	pt^ := (pData^ / 16#10) + 48 + (((pData^ / 16#10)/10)*7);
	pt:=pt+1;
	pt^ := (pData^ AND 16#0F)  + 48 + (((pData^ AND 16#0F)/10)*7);
	pt:=pt+1;

	xl:=xl+2;

	DataLen:=DataLen-1;
	pData:=pData+1;

END_WHILE

pt^:=0;
END_FUNCTION

(* POU Plant_Objects/obj_CIR, ST *)
FUNCTION_BLOCK obj_CIR

(* === CIRCOLATORE STANDARD ===
   v1.0[16/04/15] - Versioning
   v1.1[11/08/15] - Added status reconstruction
*)
VAR CONSTANT
	SampleNr		: BYTE := 120;	(* 1 minute of observation *)
END_VAR
VAR_INPUT
	(* Settings *)
	ID				: BYTE;
	ExtStatus		: BOOL;	(* TRUE: external status signal input available, FALSE: no external status input *)

	(* Physical inputs (Force) *)
	CIR_RUN_REQ		: BOOL; (* External run request (no heat or cold requested) *)
	CIR_STOP_REQ	: BOOL; (* External stop request (has priority over RUN signals!) *)

	(* Physical inputs (Feedback) *)
	Pump_AL			: BOOL; (* Pump Alarm *)
	Pump_ST			: BOOL; (* Pump Status *)
	Pump_AUTO		: BOOL; (* Pump Auto/Manual *)

	(* Controls *)
	OnOff			: BOOL;	(* On/Off from chrono *)
	InitOK			: BOOL;

	(* Timings *)
	OnDelay		:	TIME;	(* Switch on delay *)
	OffDelay	:	TIME;	(* Switch off delay *)

	(* Input temperature needed if no real feedback about status is available *)
	Tprobe		:	INT;
END_VAR
VAR_OUTPUT
	CIR_EN			: BOOL;

	Ctrl_Run		: BOOL;		(* Logical status of the device: 0: Not running (switched off), 1: running *)
	Run				: BOOL;		(* Real status *)

	Status_Log		: WORD;
	Status_Vis		: DWORD;
END_VAR
VAR
	CIR_AUTO	: 	BOOL; (* Auto/Manual input signal *)
	Pump_En		:	BOOL;

	(* Filters *)
	fPump_ST	: 	FLT_TAP := (INITEV:=FALSE);
	fPump_En	:	FLT_EVENT;
	fCIR_AUTO	:	FLT_TAP;
	fStatus		:	FLT_EVENT;
	fStatusFault:	BOOL;

	(* Timer manage switch on/off delay *)
	Delay		: 	TONOF;

	(* Alarm and Warning counters *)
	AlarmCtr	:	BYTE;
	WarningCtr	:	BYTE;

	(* Filers on alarms and faults *)
	AlarmHw		:	FLT_TAP := (INITEV:=FALSE);

	(* Variables for status reconstruction *)
	aTprobe		:	ARRAY [1..SampleNr] OF INT;
	sample		:	BYTE;
	Tmean		:	INT;
	sum			:	INT;
	i			:	BYTE;
END_VAR
Init();

StatusRebuild();
(* Check alarms and warnings *)
CheckFault();

PumpManager();

IF AlarmCtr>0 THEN
	Status_Log := 2;
	Status_Vis := COLOR_RED;
ELSIF WarningCtr>0 OR fPump_ST.OUT THEN
	Status_Log := 1;
	Status_Vis := COLOR_YELLOW;
ELSE
	Status_Log := 0;
	Status_Vis := COLOR_GREEN;
END_IF

Lamp.UpdateStatus(obj_Status := Status_Log);
END_FUNCTION_BLOCK
ACTION AddLogData:
Logger.s1:=INSERT('&CIR=',BYTE_TO_STRING(ID),4);
IF ID<10 THEN Logger.s1:=INSERT(Logger.s1,'0',4); END_IF

Logger.s1:=CONCAT(Logger.s1,SEL(Pump_En,'0','100'));
Logger.s1:=CONCAT(Logger.s1,';');
Logger.s1:=CONCAT(Logger.s1,WORD_TO_STRING(Status_Log));
Logger.s1:=CONCAT(Logger.s1,';');
Logger.s1:=CONCAT(Logger.s1,SEL(CIR_RUN_REQ,'0','100'));
Logger.s1:=CONCAT(Logger.s1,';');
Logger.s1:=CONCAT(Logger.s1,SEL(CIR_STOP_REQ,'0','100'));


ADDSTRING(ADR(Logger.TData), ADR(Logger.s1), Logger.TLen);
END_ACTION
ACTION CheckFault:
(*** ALARMS ***)

(* Hardware alarm (physical input *)
AlarmHw(IN:=Pump_AL);

IF AlarmHw.EVH THEN
	LogEv(EL_Alarm,EO_CIR,ID,3,'');
	AlarmCtr := AlarmCtr + 1;
END_IF

IF AlarmHw.EVL THEN
	LogEv(EL_Log,EO_CIR,ID,4,'');
	AlarmCtr := SEL(AlarmCtr=0, AlarmCtr-1, 0);
END_IF

IF ExtStatus THEN
	fPump_ST(IN:=(Pump_ST<>CIR_EN));

	IF fPump_ST.EVH THEN
		IF Pump_AUTO THEN
			LogEv(SEL(Pump_ST,EL_Alarm,EL_Wrn),EO_CIR,ID,SEL(Pump_ST,5,6),'');
		ELSE
			LogEv(EL_Wrn,EO_CIR,ID,SEL(Pump_ST,1,2),'');
		END_IF
	END_IF

ELSE
	fPump_ST(IN:=fStatusFault);

	IF fPump_ST.EVH THEN
		IF Pump_AUTO THEN
			LogEv(SEL(OnOff,EL_Alarm,EL_Wrn),EO_CIR,ID,SEL(OnOff,5,6),'');
		ELSE
			LogEv(EL_Wrn,EO_CIR,ID,SEL(OnOff,1,2),'');
		END_IF
	END_IF
END_IF
END_ACTION
ACTION Init:
IF NOT InitOK THEN

	Delay.PT_OF := SEL(OffDelay=T#0ms, OffDelay, Plant_CirOffDelay);
	Delay.PT_ON := SEL(OnDelay=T#0ms, OnDelay, Plant_CirOnDelay) + WORD_TO_TIME(1000*ID);

	Pump_En := FALSE;

	InitOK := TRUE;

END_IF
END_ACTION
ACTION PumpManager:
(* Verify if in Auto or Manual mode *)
fCIR_AUTO(IN:=Pump_AUTO);

IF fCIR_AUTO.EVH THEN
	LogEv(EL_Log,EO_CIR,ID,8,'CIR_Auto');
	WarningCtr := SEL(WarningCtr=0, WarningCtr-1,0);
END_IF

(* Manual -> Keep switched on *)
IF fCIR_AUTO.EVL THEN
	LogEv(EL_Wrn,EO_CIR,ID,7,'CIR_Manual');
	WarningCtr := WarningCtr + 1;

	(* Switch on pump *)
	Pump_En := TRUE;
END_IF

(* Verify if OnOff is changed *)
Ctrl_Run := OnOff;

(* Check switch on or switch off delay *)
Delay(IN:=Ctrl_Run);

(* Do these instructions only if in AUTO mode *)
IF Pump_AUTO THEN
	(* If priority request *)
	IF CIR_STOP_REQ THEN Pump_En := FALSE;
	ELSIF CIR_RUN_REQ THEN Pump_En := TRUE;
	ELSE Pump_En := Delay.OUT;
	END_IF

	(* Set RUN signal (for external objects) *)
	IF AlarmHw.OUT THEN
		Run:=FALSE;
	ELSE
		Run:=Pump_En;
	END_IF
END_IF

(* Set value on physical outuput! *)
CIR_EN := Pump_En;
END_ACTION
ACTION StatusRebuild:
IF NOT ExtStatus THEN
	(* Check every 20 seconds *)
	IF  sample<sampleNr THEN
	
		aTprobe[sample] := Tprobe;
		sample := sample + 1;
	
	ELSE
	
		SHIFT_ARRAY(ADR(aTprobe),SampleNr);
	
		FOR i:=1 TO SampleNr BY 1 DO
			sum := sum + aTprobe[i];
		END_FOR
	
		Tmean := sum/SampleNr;
	
		(* CIR should be on but revealed temperature is decreasing *)
		IF OnOff AND (Tprobe<aTprobe[1]) THEN
			fStatusFault := TRUE;
		ELSE
			fStatusFault := FALSE;
		END_IF
	
		(* CIR should be off but revealed temperature is increasing *)
		IF NOT OnOff AND (Tprobe>aTprobe[1]) THEN
			fStatusFault := TRUE;
		ELSE
			fStatusFault := FALSE;
		END_IF
	END_IF
END_IF
END_ACTION

(* POU Utils Functions/TONOF, ST *)
FUNCTION_BLOCK TONOF
VAR_INPUT
	IN		: BOOL;
	PT_ON	: TIME; (* time to pass, before OUT is set *)
	PT_OF	: TIME; (* time to pass, before OUT is reset *)
END_VAR
VAR_OUTPUT
	OUT		: BOOL;
END_VAR
VAR
	timer	: TON;
END_VAR
IF IN<>OUT THEN
	timer(IN:=TRUE,PT:=SEL(IN,PT_OF,PT_ON));
	IF timer.Q THEN OUT:=IN; END_IF
ELSE
	timer(IN:=FALSE);
END_IF
END_FUNCTION_BLOCK

(* POU Plant_Objects/obj_CRON_EDITOR, ST *)
FUNCTION_BLOCK obj_CRON_EDITOR
(* === EDITOR CRONOGRAFO ===
   v1.0[16/04/15] - Versioning
   v1.1[19/05/15] - Create empty profile when not found
*)
VAR_INPUT

	(* Common selections *)
	CN_Sel:			BYTE:=1;
	CN_Act:			BYTE;
	CN_YSel:		WORD:=2015;
	CN_YAct:		WORD;

	(* Profile editor *)
	PR_Sel: 		BYTE:=1;
	PR_Act:			BYTE;
	PR_TT:			REAL;
	PR:				typ_Cron_Profile;
	(* Profile signals *)
	PR_Load:		BOOL;
	PR_Save:		BOOL;

	(* Calendar editor *)
	CA_Sel:			BYTE:=1; (* Calendar month selected *)
	CA_Act:			BYTE;    (* Calendar month active *)
	CA_DayF:		BYTE:=0;
	CA_DayL:		BYTE:=31;
	CA_TPR:			BYTE;
	CA:				typ_Cron_Calendar; (* Only used for first 32 entries *)
	(* Calendar signals *)
	CA_Load:		BOOL;
	CA_Save:		BOOL;

	(* Jolly editor *)
	JL:				ARRAY[0..9] OF typ_Cron_Jolly;
	(* Jolly signals *)
	JL_Load:		BOOL;
	JL_Save:		BOOL;

END_VAR
VAR_OUTPUT
	Message		: STRING;
END_VAR
VAR
	sFileName	: STRING;
	sFileMode	: STRING;
	hFile		: DWORD;
	Buf			: ARRAY[0..512] OF BYTE; (* AVOID THIS!! *)

	i			: WORD;
	ver			: BYTE;
	r1			: BOOL;
	r2			: DWORD;

END_VAR
IF PR_Load THEN PR_Load_Exe(); PR_Load:=FALSE; END_IF
IF PR_Save THEN PR_Save_Exe(); PR_Save:=FALSE; END_IF
IF CA_Load THEN CA_Load_Exe(); CA_Load:=FALSE; END_IF
IF CA_Save THEN CA_Save_Exe(); CA_Save:=FALSE; END_IF
IF JL_Load THEN JL_Load_Exe(); JL_Load:=FALSE; END_IF
IF JL_Save THEN JL_Save_Exe(); JL_Save:=FALSE; END_IF
END_FUNCTION_BLOCK
ACTION CA_Load_Exe:
sFileMode:='r';
FileOpen();

IF hFile<>0 THEN

	(* Read calendar month *)
	FOR i := 0 TO 31 DO
		r1:=SysFileSetPos(File:=hFile, Pos:=(1024 + ((CA_Sel-1)*32 + i)*4));
		r2:=SysFileRead(File:=hFile, Buffer:=ADR(CA.Profile[i]), Size:=1);
	END_FOR

	(* Close file *)
	SysFileClose(File:=hFile);

	(* Validate data *)
	CA_Act :=CA_Sel;
	CN_Act :=CN_Sel;
	CN_YAct:=CN_YSel;

	Message:='Calendar load OK';

END_IF
END_ACTION
ACTION CA_Save_Exe:
sFileMode:='a';
FileOpen();

IF hFile<>0 THEN

	(* Write calendar month *)
	FOR i := 0 TO 31 DO
		r1:=SysFileSetPos(File:=hFile, Pos:=(1024 + ((CA_Sel-1)*32 + i)*4));
		r2:=SysFileGetPos(hFile);
		r2:=SysFileWrite(File:=hFile, Buffer:=ADR(CA.Profile[i]), Size:=1);
	END_FOR

	(* Close file *)
	SysFileClose(File:=hFile);

	Message:='Calendar save OK';

END_IF
END_ACTION
ACTION FileOpen:
(* Create current filename 'yyyyCRnn.DAT' *)
sFileName:=CONCAT(FilesPath,WORD_TO_STRING(CN_YSel));
sFileName:=CONCAT(STR1:=sFileName, STR2:='CR');
IF CN_Sel<10 THEN
sFileName:=CONCAT(STR1:=sFileName, STR2:='0');
END_IF
sFileName:=CONCAT(STR1:=sFileName, STR2:=BYTE_TO_STRING(CN_Sel));
sFileName:=CONCAT(STR1:=sFileName, STR2:='.DAT');

(* Check file version and size! *)
(* ... *)

(* Open data file *)
hFile:=SysFileOpen(FileName:=sFileName, Mode:='r');

(* File not found *)
IF hFile=0 THEN
	Message:='File not found - created empty file';
	(* Create empty file *)
	hFile:=SysFileOpen(FileName:=sFileName, Mode:='w');
	MEMCLR(pDestinationAddress:=ADR(Buf), BytesToClear:=SIZEOF(Buf));
	FOR i := 0 TO 10239 BY 512 DO
		SysFileWrite(File:=hFile, Buffer:=ADR(Buf), Size:=512);
	END_FOR
	Buf[0]:=1;
	SysFileSetPos(File:=hFile, Pos:=0);
	SysFileWrite(File:=hFile, Buffer:=ADR(Buf), Size:=1);
END_IF

(* Close file *)
SysFileClose(File:=hFile);

(* Open data file *)
hFile:=SysFileOpen(FileName:=sFileName, Mode:=sFileMode);
END_ACTION
ACTION JL_Load_Exe:
sFileMode:='r';
FileOpen();

IF hFile<>0 THEN

	(* Read jolly *)
	r1:=SysFileSetPos(File:=hFile, Pos:=512);
	r2:=SysFileRead(File:=hFile, Buffer:=ADR(JL), Size:=SIZEOF(JL));

	(* Close file *)
	SysFileClose(File:=hFile);

	(* Validate data *)
	CN_Act:=CN_Sel;
	CN_YAct:=CN_YSel;

	Message:='Jolly load OK';

END_IF
END_ACTION
ACTION JL_Save_Exe:
sFileMode:='a';
FileOpen();

IF hFile<>0 THEN

	(* Write selected profile *)
	r1:=SysFileSetPos(File:=hFile, Pos:=512);
	r2:=SysFileWrite(File:=hFile, Buffer:=ADR(JL), Size:=SIZEOF(JL));

	(* Close file *)
	SysFileClose(File:=hFile);

	Message:='Jolly save OK';

END_IF
END_ACTION
ACTION PR_Load_Exe:
sFileMode:='r';
FileOpen();

IF hFile<>0 THEN

	(* Read selected profile *)
	r1:=SysFileSetPos(File:=hFile, Pos:=(3072 + 512*PR_Sel));
	r2:=SysFileRead(File:=hFile, Buffer:=ADR(PR), Size:=SIZEOF(PR));

	(* Close file *)
	SysFileClose(File:=hFile);

	(* Validate data *)
	PR_Act:=PR_Sel;
	CN_Act:=CN_Sel;
	CN_YAct:=CN_YSel;

	Message:='Profile load OK';

END_IF
END_ACTION
ACTION PR_Save_Exe:
sFileMode:='a';
FileOpen();

IF hFile<>0 THEN

	(* Write selected profile *)
	r1:=SysFileSetPos(File:=hFile, Pos:=(3072 + 512*PR_Sel));
	r2:=SysFileWrite(File:=hFile, Buffer:=ADR(PR), Size:=SIZEOF(PR));

	(* Close file *)
	SysFileClose(File:=hFile);

	Message:='Profile save OK';

END_IF
END_ACTION

(* POU Plant_Objects/obj_CRONTER, ST *)
FUNCTION_BLOCK obj_CRONTER
(* === THERMOSTAT ===
   v1.0[30/07/15] - Versioning
*)
VAR_INPUT
	(* Settings *)
	ID			: BYTE;		(* Index of instanced object *)

	InitOK		: BOOL;
	Alarm		: BOOL;
	Warning		: BOOL;

	Profile		: typ_Cron_Profile; 				(* Profilo attivo *)
	ProfileNr	: BYTE;								(* Indice profilo attivo *)
	CalendarIdx : WORD;								(* Indice calendario attivo *)
	Jolly		: ARRAY[0..9] OF typ_Cron_Jolly;	(* Jolly attivi *)

	Temperature	: INT;
	Local_MaxRunTAmb	:	INT;					(* Local maximum environment temperature, NOT "TAMB" *)


	Histeresys:INT; (* isteresi per la ripartenza del Comando ON*)


END_VAR
VAR_IN_OUT
END_VAR
VAR_OUTPUT
	SetPoint		: INT;
	Run				: BOOL;
	AntifreezeForce	: BOOL;

	(* Status *)
	Status_Log		: BYTE;
	Status_Vis 		: DWORD;
END_VAR
VAR
	Buf: 	ARRAY[0..512] OF BYTE; (* AVOID THIS!! *)
	hFile: 	DWORD;
	sFile: 	STRING;
	sFile2: STRING;

	i:		WORD;
	t1:		DWORD;
	t2:		BOOL;

END_VAR
(* Check initialization *)
IF NOT InitOK THEN Init(); END_IF

(* Check Temperature *)
IF Temperature < 400(*Local_MaxRunTAmb*) THEN

	(* LOCAL environment temperature lower than maximum allowed -> Proceed with SetPoint adjustment *)
	(* Chrono *)
	IF CalendarIdx<>Sys.Time_CT_Day THEN DB_Load(); END_IF
	SetPoint:=Profile.Setpoint[Sys.Time_CT_Quarter];

	(* Check jolly *)
	FOR i := 0 TO 9 DO
		IF ( DT_TO_DWORD(Jolly[i].Start)>0  AND Jolly[i].End>Jolly[i].Start AND
		     Jolly[i].Start<=Sys.Time_CT_DT AND Jolly[i].End>Sys.Time_CT_DT ) THEN
				SetPoint:=Jolly[i].Temp;
		END_IF
	END_FOR

(*
	IF SetPoint < 180 THEN
		(* Switch off the device *)
		Run := FALSE;
	ELSE
		(* Set according to feedback T - Histeresys of 1°C *)
		IF Temperature >= (SetPoint + 5) THEN
			Run := FALSE;
		ELSIF Temperature <= (SetPoint - 5) THEN
			Run := TRUE;
		END_IF

		(* Between "SetPoint-5" and "SetPoint+5" last state (ON or OFF) of "Run" is kept	*)
	END_IF
*)
(*	IF SetPoint>0 THEN Run := TRUE;
	ELSIF SetPoint=0 THEN Run := FALSE;
	END_IF *)

		IF Temperature >= (SetPoint) THEN
			Run := FALSE;
		ELSIF Temperature <= (SetPoint - Histeresys) THEN
			Run := TRUE;
		END_IF




ELSE
	(* Environment overtemperature: stop heating -> Stop device *)
	Run := FALSE;
END_IF

(* Freeze warning: Switch on and heat! *)
(*IF Temperature < Plant_AntiFreezeTAmb THEN AntifreezeForce := TRUE;
ELSE AntifreezeForce := FALSE;
END_IF*)



(* Status color *)
   IF Alarm   THEN Status_Log:=2; Status_Vis:=COLOR_RED;
ELSIF Warning THEN Status_Log:=1; Status_Vis:=COLOR_YELLOW;
              ELSE Status_Log:=0; Status_Vis:=COLOR_GREEN;
			  END_IF
END_FUNCTION_BLOCK
ACTION AddLogData:
Logger.s1:=INSERT('&THER=',BYTE_TO_STRING(ID),5);
IF ID<10 THEN Logger.s1:=INSERT(Logger.s1,'0',5); END_IF

Logger.s1:=CONCAT(Logger.s1,INT_TO_STRING(SetPoint));			Logger.s1:=CONCAT(Logger.s1,';');

Logger.s1:=CONCAT(Logger.s1,WORD_TO_STRING(Status_Log));
ADDSTRING(ADR(Logger.TData), ADR(Logger.s1), Logger.TLen);
END_ACTION
ACTION DB_Create:
(* Create empty file *)
hFile:=SysFileOpen(FileName:=sFile, Mode:='w');

MEMCLR(pDestinationAddress:=ADR(Buf), BytesToClear:=SIZEOF(Buf));
FOR i := 0 TO 10239 BY 512 DO
	t1:=SysFileWrite(File:=hFile, Buffer:=ADR(Buf), Size:=512);		(* Clear created file (all bytes 0) *)
END_FOR
Buf[0]:=1;
t2:=SysFileSetPos(File:=hFile, Pos:=0);
t1:=SysFileWrite(File:=hFile, Buffer:=ADR(Buf), Size:=1);
SysFileClose(File:=hFile);
END_ACTION
ACTION DB_Load:
DB_SetName();

(* Open data file *)
hFile:=SysFileOpen(FileName:=sFile, Mode:='r');

(* File not found *)
IF hFile=0 THEN
	Warning:=TRUE;
	LogEv(EL_Wrn,EO_CRON,ID,1,'No_data_file');
	DB_Create();
	(* Reopen file *)
	hFile:=SysFileOpen(FileName:=sFile, Mode:='r');
	IF hfile=0 THEN
		Alarm:=TRUE;
		LogEv(EL_Alarm,EO_CRON,ID,3,'Filesystem_error');
		RETURN;
	END_IF
END_IF

(* Check version *)
SysFileRead(File:=hFile, Buffer:=ADR(Buf), Size:=1);
IF Buf[0]<>1 THEN
	IF NOT Alarm THEN
		Alarm:=TRUE;
		LogEv(EL_Alarm,EO_CRON,ID,2,'Bad_data_version');
	END_IF
	SysFileClose(File:=hFile);
	RETURN;
END_IF

(* Read Jolly data *)
t2:=SysFileSetPos(File:=hFile, Pos:=512);
t1:=SysFileRead(File:=hFile, Buffer:=ADR(Jolly), Size:=SIZEOF(Jolly));
(* Read active profile index *)
CalendarIdx:=Sys.Time_CT_Day;
t2:=SysFileSetPos(File:=hFile, Pos:=(1024+4*CalendarIdx));
t1:=SysFileRead(File:=hFile, Buffer:=ADR(ProfileNr), Size:=SIZEOF(ProfileNr));
(* Read active profile *)
t2:=SysFileSetPos(File:=hFile, Pos:=(3072+512*ProfileNr));
t1:=SysFileRead(File:=hFile, Buffer:=ADR(Profile), Size:=SIZEOF(Profile));

(* Close file and validate data *)
SysFileClose(File:=hFile);
END_ACTION
ACTION DB_SetName:
(* Create current filename 'yyyyCRnn.DAT' *)
sFile:=CONCAT(FilesPath,WORD_TO_STRING(Sys.Time_Year));
sFile:=CONCAT(STR1:=sFile, STR2:='CR');
IF ID<10 THEN
sFile:=CONCAT(STR1:=sFile, STR2:='0');
END_IF
sFile:=CONCAT(STR1:=sFile, STR2:=BYTE_TO_STRING(ID));
sFile:=CONCAT(STR1:=sFile, STR2:='.DAT');
END_ACTION
ACTION Init:
DB_Load();
InitOK:=TRUE;
END_ACTION

(* POU Plant_Objects/obj_CTL, ST *)
FUNCTION_BLOCK obj_CTL
(* === PULSE VOLUME COUNTER ===
   v1.0[16/04/15] - Versioning
*)
VAR_INPUT
	(* Settings *)
	ID				: BYTE;	(* Index of instanced object *)
	Peso			: DWORD;
	(* Physical inputs *)
	CTL_ST			: BOOL;
END_VAR
VAR_IN_OUT
	COUNT			: DWORD;
END_VAR
VAR_OUTPUT
	(* Status *)
	Status_Log		: BYTE;
END_VAR
VAR
	Filter			: FLT_TAP := ( INITEV:=FALSE );
	Filter01			: FLT_TAP := ( INITEV:=FALSE );
	Timer			: TON;
	TCount			: DWORD;
	TCount01		: DWORD;
	i				: DWORD;

	TempoSicurezzaPerdita: DINT;
	TimerConataLitriPerdita:TOF;


	MorenoTest: BOOL;
	erroreTest: BOOL;
END_VAR

VAR_INPUT RETAIN
	LimiteMaxPerdita: INT;
END_VAR
(* Execute timer *)
Timer(IN:=NOT Timer.Q, PT:=T#60m);

(* Execute filter on counter status *)
Filter(IN:=CTL_ST);
Filter01(IN:=CTL_ST);


(*

(* Count event *)
IF Filter.EVH THEN
	COUNT:=COUNT+Peso;

	TCount:=TCount+1;
	(* Check flow rate *)
	IF TCount>=Plant_MaxWaterLoss THEN


		i:=(TCount*TIME_TO_DWORD(Timer.PT))/TIME_TO_DWORD(Timer.ET);	(* Estimated mc per hour *)
		i:= i * Peso;

		(* NB The weight is multiplied by 10 -> Need to divide it by 10 server side *)
		LogEv(EL_AlarmStop,EO_CTL,ID,1,DWORD_TO_STRING(i));
		Status_Log:=2;

		TCount:=0;
		Timer(IN:=FALSE);
	END_IF
END_IF
(* Check timer *)
IF Timer.Q THEN
	TCount:=0;							(* One hour is elapsed *)
	IF TCount<Plant_MaxWaterLoss THEN
		Status_Log:=0;
	END_IF
END_IF

*)


(*** calcolo del tempo del contalitri minimo per la segnalazione dell'allarme perdita *****)

(* il limiteMAXPerdita è espresso in l/h con n.1 decimale, Quindi dividendolo per il peso dell'impulso e per 60minuti, otteniamo
quanto tempo deve passare minimo fra un impulsao e l'altro *)

LimiteMaxPerdita:=LIMIT(LimiteMaxPerdita,10,LimiteMaxPerdita+1);
TempoSicurezzaPerdita:=3600000/((LimiteMaxPerdita/peso)); (* espresso in ms *)

IF Filter01.EVH THEN
(*	COUNT:=COUNT+Peso; *)

	TCount01:=TCount01+1;
	IF TimerConataLitriPerdita.Q AND NOT erroreTest THEN

		(* NB The weight is multiplied by 10 -> Need to divide it by 10 server side *)

		LogEv(EL_AlarmStop,EO_CTL,ID,1,CONCAT('LimiteMAXPerdita_l/h>',DWORD_TO_STRING(LimiteMaxPerdita/10)));
		Status_Log:=2;

		erroreTest:=TRUE;
		TimerConataLitriPerdita(IN:=FALSE, PT:= t#1s, Q=> , ET=> );
	END_IF


	IF NOT TimerConataLitriPerdita.Q AND erroreTest THEN
		erroreTest:=FALSE;
		TCount01:=0;
		Status_Log:=0;
	END_IF

END_IF





TimerConataLitriPerdita(IN:=Filter01.EVH, PT:= DINT_TO_TIME(TempoSicurezzaPerdita), Q=> , ET=> );
END_FUNCTION_BLOCK
ACTION AddLogData:
Logger.s1:=INSERT('&CTL=',BYTE_TO_STRING(ID),4);
IF ID<10 THEN Logger.s1:=INSERT(Logger.s1,'0',4); END_IF

Logger.s1:=CONCAT(Logger.s1,DWORD_TO_STRING(COUNT));			Logger.s1:=CONCAT(Logger.s1,';');

Logger.s1:=CONCAT(Logger.s1,WORD_TO_STRING(Status_Log));
ADDSTRING(ADR(Logger.TData), ADR(Logger.s1), Logger.TLen);
END_ACTION

(* POU Plant_Objects/obj_MBUS, ST *)
FUNCTION_BLOCK obj_MBUS
(* === M-BUS PROTOCOL INTERFACE ===
   v1.0[16/03/15] - Added interface errors
*)
VAR_INPUT
	(* Settings *)
	ID				: BYTE;
	COM				: BYTE;
	BAUDRATE		: COM_BAUDRATE;
	(* Interface *)
	MBus 			: typMBus;
	MBus_Master 	: FbMBusMaster;
END_VAR
VAR_OUTPUT
	(* Status *)
	Status_Log		: BYTE;
	Status_Vis 		: DWORD;
END_VAR
VAR
	Alarm			: FLT_EVENT;
END_VAR
MBus_Master( bCOMPORT:=COM , enumBAUDRATE:=BAUDRATE , utMBus:=MBus );

(* Check status *)
Alarm(IN:=(MBus.bCOM_ERROR<>0));
IF Alarm.EVH THEN
	LogEv(EL_Alarm,EO_MBUS,ID,1,BYTE_TO_STRING(MBus.bCOM_ERROR));
END_IF
IF Alarm.EVL THEN
	LogEv(EL_Log,EO_MBUS,ID,2,'MBUS_OK');
END_IF

(* Log/visu status *)
   IF Alarm.IN   					THEN Status_Log:=2; Status_Vis:=COLOR_RED;
ELSIF (MBus.bL1_ERROR AND 16#1F)<>0 THEN Status_Log:=1; Status_Vis:=COLOR_YELLOW;
  				 					ELSE Status_Log:=0; Status_Vis:=COLOR_GREEN;
END_IF
END_FUNCTION_BLOCK

(* POU Plant_Objects/obj_MBUS_CTB_SHARKY775, ST *)
FUNCTION_BLOCK obj_MBUS_CTB_SHARKY775
(* === M-BUS CONTABILIZER SHARKY 775 ===
   v1.0[16/03/15] - Error management
*)
VAR_INPUT
	(* Settings *)
	ID				: BYTE;
	ADDRESS			: DWORD;
	Refresh_Period	: TIME:=t#3m;
	(* Controls *)
	Refresh_Auto	: BOOL:=TRUE; (* Enable automatic refresh *)
	Refresh_Now		: BOOL; 	  (* Force an immediate refresh *)
END_VAR
VAR_IN_OUT
	(* Interface *)
	MBUS			: obj_MBUS;
END_VAR
VAR_OUTPUT
	M1				: FbMBus_Heat;
	(* Status *)
	Status_Log		: BYTE;
	Status_Vis 	 	: DWORD;
END_VAR
VAR
	dly 	 	: TON := (PT:=t#5s);
	M1_Start	: BOOL;

	init_st		: BOOL;
	bus_st0		: BYTE;
	dev_st0		: BYTE;

(*	S1			: FbMBusSend;
	S1_Start	: BOOL;*)
(*	C1			: FbUnitConverter; *)

END_VAR
(* Auto refresh timer *)
dly(IN:=NOT (dly.Q OR Refresh_Now OR (NOT Refresh_Auto)));
(* Trigger refresh *)
IF dly.Q OR Refresh_Now THEN
	dly.PT:=Refresh_Period;
	Refresh_Now:=FALSE;
	(* Start reading *)
	M1.dwAdr:= ADDRESS;
	M1.xSND_NKE:=TRUE;
	M1_Start:=TRUE;
END_IF

(* Contabilizer module *)
M1(	utMBus:=MBUS.MBus, xStart:=M1_Start );

(* Extra actions *)
(*C1( utMBus:=MBUS.MBus, xStart:=C1_Start );*)

(* Check status *)
IF NOT init_st OR M1.bError<>bus_st0 OR M1.utMBInfo.bMStatus<>dev_st0 THEN
	init_st:=TRUE;
	bus_st0:=M1.bError; dev_st0:=M1.utMBInfo.bMStatus;
	IF bus_st0<>0 THEN
		LogEv(EL_Alarm,EO_CTB,ID,2,BYTE_TO_STRING(bus_st0));
		Status_Log:=2; Status_Vis:=COLOR_RED;
	ELSE
		IF dev_st0<>0 THEN
			Status_Log:=2; Status_Vis:=COLOR_RED;
			CASE dev_st0 OF
				16#08: LogEv(EL_Alarm,EO_CTB,ID,10,'C-1');
				16#04: LogEv(EL_Alarm,EO_CTB,ID,10,'E-8');
				16#28: LogEv(EL_Alarm,EO_CTB,ID,10,'E-4');
				16#50: LogEv(EL_Alarm,EO_CTB,ID,10,'E-1');
				16#70: LogEv(EL_Alarm,EO_CTB,ID,10,'E-7');
				16#84: LogEv(EL_Alarm,EO_CTB,ID,10,'E-9');
				16#B0: LogEv(EL_Wrn  ,EO_CTB,ID,10,'E-3');
				16#D0: LogEv(EL_Wrn  ,EO_CTB,ID,10,'E-6');
				16#F0: LogEv(EL_Alarm,EO_CTB,ID,10,'Leak');
				16#10: LogEv(EL_Wrn  ,EO_CTB,ID,10,'E-5'); Status_Log:=1; Status_Vis:=COLOR_YELLOW;
			ELSE
				LogEv(EL_Alarm,EO_CTB,ID,10,BYTE_TO_STRING(dev_st0));
			END_CASE
		ELSE
			Status_Log:=0; Status_Vis:=16#20F020;
			LogEv(EL_Log,EO_CTB,ID,1,'');
		END_IF
	END_IF
END_IF

Lamp.obj_Status := Status_Log;
Lamp.UpdateStatus();
END_FUNCTION_BLOCK
ACTION AddLogData:
Logger.s1:=INSERT('&CTB=',BYTE_TO_STRING(ID),4);
IF ID<10 THEN Logger.s1:=INSERT(Logger.s1,'0',4); END_IF

Logger.s1:=CONCAT(Logger.s1,M1.utFTemp.Value);		Logger.s1:=CONCAT(Logger.s1,';');
Logger.s1:=CONCAT(Logger.s1,M1.utRTemp.Value);		Logger.s1:=CONCAT(Logger.s1,';');
Logger.s1:=CONCAT(Logger.s1,M1.utFlow.Value);		Logger.s1:=CONCAT(Logger.s1,';');
Logger.s1:=CONCAT(Logger.s1,M1.utPower.Value);		Logger.s1:=CONCAT(Logger.s1,';');
Logger.s1:=CONCAT(Logger.s1,M1.utEnergy.Value);		Logger.s1:=CONCAT(Logger.s1,';');

Logger.s1:=CONCAT(Logger.s1,BYTE_TO_STRING(Status_Log));
ADDSTRING(ADR(Logger.TData), ADR(Logger.s1), Logger.TLen);
END_ACTION

(* POU Plant_Objects/obj_MODBUS, ST *)
FUNCTION_BLOCK obj_MODBUS
(* === MODBUS PROTOCOL INTERFACE ===
   v1.1[19/06/15] - Added new VARS allocation and searching
*)
VAR CONSTANT
	VARS_Max	: BYTE := 32;
END_VAR
VAR_INPUT
	(* Settings *)
	ID			: BYTE;
	COM			: BYTE;
	BAUDRATE	: COM_BAUDRATE;
	RS485		: BOOL := FALSE;

	(* Interface *)
	MB_MASTER	: MODBUS_EXTENDED_MASTER;
	MB_Start	: BOOL;
	MB_Query	: typModbusExtendedQuery;
	MB_Resp		: typModbusResponse;
	MB_Lock		: BOOL;

	(* Variables management *)
	VARS_En		: BOOL;
	VARS		: ARRAY [0..VARS_Max] OF typ_MODBUS_VAR;
	VARS_Check	: BOOL;
	VARS_Alarm	: BOOL;

	(* Variables allocation *)
	VAR_Pointer : POINTER TO ARRAY[0..99] OF WORD;
	VAR_Cfg		: POINTER TO typ_MODBUS_VAR;
END_VAR
VAR_OUTPUT
	(* Status *)
	Status_Log	: BYTE;
	Status_Vis	: DWORD;
END_VAR
VAR
	sta         : BYTE :=0;
	i			: BYTE;
	j			: BYTE;
	Alarm		: FLT_EVENT;
	
	VarTmr		: TON := (PT:=T#1s);
	VarSta		: BYTE; (* Status *)
	VarCnt		: BYTE; (* Scan counter *)
	VarRetry	: BYTE;
	VarAlarm	: BYTE; (* Last variable with errors *)
END_VAR
MB_MASTER(ENABLE:=TRUE,	ASCII_Mode:=FALSE, bCOM_PORT:=COM, cbCOM_BAUDRATE:=BAUDRATE, cpCOM_PARITY:=PARITY_NO,
		csCOM_STOPBITS:=STOPBITS_1,	cbsCOM_BYTESIZE:=BS_8, cfCOM_FLOW_CONTROL:=SEL(RS485,NO_FLOW_CONTROL,HALFDUPLEX),
		tTIME_OUT:=t#250ms,	StartFunction:=MB_Start, ExtQuery:=MB_Query, Response:=MB_Resp);

(* Process variable management *)
IF VARS_En THEN VARS_Process(); END_IF

(* Check status *)
Alarm(IN:=(MB_MASTER.bInterfaceError<>0));
IF Alarm.EVH THEN
	LogEv(SEL(MB_MASTER.bInterfaceError<>3,EL_Wrn,EL_Alarm),EO_MODBUS,ID,1,BYTE_TO_STRING(MB_MASTER.bInterfaceError));
END_IF
IF Alarm.EVL THEN								(* Trigger a fall edge: MODBUS back working *)
	LogEv(EL_Log,EO_MODBUS,ID,2,'MODBUS_OK');
END_IF

(* Log/visu status *)
   IF Alarm.IN   THEN Status_Log:=2; Status_Vis:=COLOR_RED;
ELSIF Vars_Alarm THEN Status_Log:=1; Status_Vis:=COLOR_YELLOW;
  				 ELSE Status_Log:=0; Status_Vis:=COLOR_GREEN;
END_IF
END_FUNCTION_BLOCK
ACTION VAR_Search:
(* Search VAR with specific pointer if not found return first free VAR
	[Last VAR is not active... used as safe area...] 
*)
j:=VARS_Max;
FOR i := 0 TO VARS_Max-1 DO
	IF VARS[i].Variable=0 AND j>i THEN j:=i; END_IF
	IF VARS[i].Variable=VAR_Pointer THEN
		VAR_Cfg:=ADR(VARS[i]);
		RETURN;
	END_IF
END_FOR
VAR_Cfg:=ADR(VARS[j]);
END_ACTION
ACTION VARS_Process:
(* Update var timers *)
VarTmr(IN:=(NOT VarTmr.Q));
IF VarTmr.Q THEN
	FOR i := 0 TO VARS_Max DO
		IF VARS[i].Refresh_Cnt>0 THEN VARS[i].Refresh_Cnt:=VARS[i].Refresh_Cnt-1; END_IF
	END_FOR
	VARS_Check:=TRUE;
END_IF


(* Process status *)
CASE VarSta OF
	0: (* === Init *)
		VarCnt:=0;
		VarSta:=1;

	1: (* === Wait check signal *)
		IF VARS_Check THEN				(* Decremented "Refresh_Cnt" *)
			VARS_Check:=FALSE;
			VarCnt:=0;
			VarSta:=2;
		END_IF

	2: (* === Check loop *)
		IF NOT (MB_Lock OR MB_Start) THEN
			WHILE VarCnt<=(VARS_Max-1) AND VarSta=2 DO
				(* Check only active vars *)
				IF VARS[VarCnt].Variable<>0 THEN			(* "Variable" is a pointer to word, so if 0 no address *)
					(* Check var auto-refresh on timer checks *)
					IF VARS[VarCnt].Refresh_Time>0 AND VARS[VarCnt].Refresh_Cnt=0 THEN
						VARS[VarCnt].Refresh_Cnt:=VARS[VarCnt].Refresh_Time;
						VarSta:=3;
					END_IF
					(* Check refresh for change or request *)
					CASE VARS[VarCnt].FunCode OF
						5,6,15,16: (* Write functions *)
							IF VARS[VarCnt].Variable_Size=1 THEN
								IF VARS[VarCnt].Variable^<>VARS[VarCnt].Variable_Mirror THEN
									VARS[VarCnt].Variable_Mirror:=VARS[VarCnt].Variable^;
									VarSta:=3;
								END_IF
							ELSE
								IF VARS[VarCnt].Variable_Mirror<>0 THEN
									VARS[VarCnt].Variable_Mirror:=0;
									VarSta:=3;
								END_IF
							END_IF
						1,2,3,4: (* Read functions *)
							IF VARS[VarCnt].Variable_Mirror<>0 THEN
								VARS[VarCnt].Variable_Mirror:=0;
								VarSta:=3;
							END_IF
					END_CASE
				END_IF
				(* Process query *)
				IF VarSta=3 THEN
					MB_Lock:=TRUE;
					MB_Query.SlaveAddress:=VARS[VarCnt].SlaveAddress;
					MB_Query.FunctionCode:=VARS[VarCnt].FunCode;
					CASE VARS[VarCnt].FunCode OF
						16#5,16#6,16#F,16#10:
							MB_Query.Read_Quantity:=0;
							MB_Query.Read_StartAddress:=0;
							MB_Query.Write_StartAddress:=VARS[VarCnt].FunAddress;
							MB_Query.Write_Quantity:=VARS[VarCnt].Variable_Size;
							IF VARS[VarCnt].Variable_Size=200 THEN
								COPY_32SWAP16(VARS[VarCnt].Variable, ADR(MB_Query.Write_Data[0]));
							ELSIF VARS[VarCnt].Variable_Size>1 THEN
								MEMCPY(VARS[VarCnt].Variable, ADR(MB_Query.Write_Data[0]), 2*VARS[VarCnt].Variable_Size);
							ELSE
								MB_Query.Write_Data[0]:=VARS[VarCnt].Variable^;
							END_IF
						16#1,16#2,16#3,16#4:
							MB_Query.Read_StartAddress:=VARS[VarCnt].FunAddress;
							IF VARS[VarCnt].Variable_Size=200 THEN MB_Query.Read_Quantity:=2; ELSE
							  MB_Query.Read_Quantity:=VARS[VarCnt].Variable_Size;
							END_IF
							MB_Query.Write_StartAddress:=0;
							MB_Query.Write_Quantity:=0;
					END_CASE
					VarRetry:=0;
					MB_Start:=TRUE;
				ELSE
					VarCnt:=VarCnt+1;
				END_IF
			END_WHILE
			(* Check loop completed -> no actions *)
			IF VarSta=2 THEN VarSta:=1; END_IF
		END_IF

	3: (* === Wait & process MB response *)
		IF NOT MB_Start THEN
			IF MB_MASTER.MB_Error=0 THEN
				CASE VARS[VarCnt].FunCode OF
					1,2,3,4:
						IF VARS[VarCnt].Variable_Size=200 THEN
							COPY_32SWAP16(ADR(MB_Resp.Data), VARS[VarCnt].Variable);
						ELSIF VARS[VarCnt].Variable_Size>1 THEN
							MEMCPY(ADR(MB_Resp.Data), VARS[VarCnt].Variable, 2*VARS[VarCnt].Variable_Size);
						ELSE
							VARS[VarCnt].Variable^:=MB_Resp.Data[0];
						END_IF
				END_CASE
				MB_Lock:=FALSE;
				(* Signal error recovery *)
				IF VARS_Alarm=TRUE AND VarCnt=VarAlarm THEN
					LogEv(EL_Wrn,EO_MODBUS,ID,5,'');
					VARS_Alarm:=FALSE;
				END_IF
				(* Next var *)
				VarCnt:=VarCnt+1;
				VarSta:=2;
			ELSE
				IF VarRetry<3 THEN
					VarRetry:=VarRetry+1;
					MB_Start:=TRUE;
				ELSE
					MB_Lock:=FALSE;
					(* Signal error *)
					IF VARS_Alarm=FALSE THEN
						LogEv(EL_Wrn,EO_MODBUS,ID,3,INT_TO_STRING(MB_MASTER.MB_Error));
						VARS_Alarm:=TRUE;
						VarAlarm:=VarCnt-1;
					END_IF
					(* Next var *)
					VarCnt:=VarCnt+1;
					VarSta:=2;
				END_IF
			END_IF
		END_IF

ELSE
	VarSta:=0;
END_CASE
END_ACTION

(* POU Plant_Objects/obj_MODBUS_CIR, ST *)
FUNCTION_BLOCK obj_MODBUS_CIR
VAR CONSTANT
	WAIT_STATE		:	BYTE := 0;
	PUMP_STATUS		:	BYTE := 1;
	PUMP_DATA		:	BYTE := 2;
	PUMP_ALARMS		:	BYTE := 3;
	PUMP_END_READ	:	BYTE := 4;
	CIR_ON_OFF		:	BYTE := 90;
	CIR_ON_OFF_CHECK:	BYTE := 91;
	CIR_END_WRITE	:	BYTE := 92;
	ERROR_STATE		:	BYTE := 100;
END_VAR
VAR_INPUT
	ID		:	BYTE;
	Address :	BYTE;		(* Pump address *)

	(* Physical inputs *)
	CIR_RUN_REQ		: BOOL; (* External run request (no heat or cold requested) *)
	CIR_STOP_REQ	: BOOL; (* External stop request (has priority over RUN signals!) *)

	Pump_AL			: BOOL; (* Alarm input signal *)
	Pump_AUTO		: BOOL;	(* Automatic/Manual input *)

	(* Controls *)
	OnOff		: 	BOOL;
	InitOK		:	BOOL;

	(* Timings *)
	OnDelay		:	TIME;
	OffDelay	:	TIME;

	(* Modbus *)
	Refresh_Now	:	BOOL;	(* Start immediately modbus state machine *)
	retryErrMax	:	BYTE := 15;
END_VAR
VAR_IN_OUT
	ModBus		:	obj_MODBUS;
END_VAR
VAR_OUTPUT
	Ctrl_Run	:	BOOL;		(* Logical status of the device: 0: Not running (switched off), 1: running *)
	Run			:	BOOL;		(* Real status *)

	Status_Log	:	WORD;
	Status_Vis	:	DWORD;
END_VAR
VAR
	Pump_En		:	WORD;

	(* Filters *)
	fPump_AL	:	FLT_TAP := (INITEV:=FALSE);
	fPump_ST	:	FLT_TAP := (INITEV:=FALSE);
	fPump_En	:	FLT_EVENT;
	fCIR_AUTO	:	FLT_TAP;
	fStatus		:	FLT_EVENT;
	fStatusFault:	BOOL;

	(* Timer manage switch on/off delay *)
	Delay		: 	TONOF;

	(* CIR data structure *)
	DataPump	:	typ_MODBUS_CIR;

	(* Modbus variables *)
	state		:	BYTE;
	retry		:	BYTE;
	retryErr	:	BYTE;
	ReadTmr		:	TON := (PT:=T#5s);
	fModbusAlr	: 	BOOL;

	(* Alarm and Warning counters *)
	AlarmCtr	:	BYTE;
	WarningCtr	:	BYTE;

	(* Filers on alarms and faults *)
	AlarmHw		:	FLT_TAP;(* := (INITEV:=FALSE);*)
	Alarm		:	FLT_EVENT := (INITEV:=FALSE);
	Inverter	:	FLT_EVENT := (INITEV:=FALSE);
	ModbusAlr	:	FLT_EVENT := (INITEV:=FALSE);

	OldAlarm	:	WORD;

	TimeOutModBus: TON;
END_VAR
Init();

(* Check alarm and warning for both pumps *)
CheckFault();

PumpManager();

(* State machine to read pump parameters *)
Stm();

IF AlarmCtr>0 THEN
	Status_Log := 2;
	Status_Vis := COLOR_RED;
ELSIF WarningCtr>0 OR fPump_ST.OUT THEN
	Status_Log := 1;
	Status_Vis := COLOR_YELLOW;
ELSE
	Status_Log := 0;
	Status_Vis := COLOR_GREEN;
END_IF

(* Update error lamp status *)
Lamp.UpdateStatus(obj_Status:=Status_Log);
END_FUNCTION_BLOCK
ACTION AddLogData:
Logger.s1:=INSERT('&CIRM=',BYTE_TO_STRING(ID),5);
IF ID<10 THEN Logger.s1:=INSERT(Logger.s1,'0',5); END_IF

(* NB If value equals 0x7FFF (32767) this means that it is not available -->> Change it to 0 *)
Logger.s1:=CONCAT(Logger.s1,WORD_TO_STRING(DataPump.PumpStatus));											Logger.s1:=CONCAT(Logger.s1,';');
Logger.s1:=CONCAT(Logger.s1,INT_TO_STRING(SEL(DataPump.PumpBoardTemp=16#7FFF,DataPump.PumpBoardTemp,0)));	Logger.s1:=CONCAT(Logger.s1,';');
Logger.s1:=CONCAT(Logger.s1,WORD_TO_STRING(SEL(DataPump.PumpVoltage=16#7FFF,DataPump.PumpVoltage,0)));		Logger.s1:=CONCAT(Logger.s1,';');
Logger.s1:=CONCAT(Logger.s1,WORD_TO_STRING(SEL(DataPump.PumpCurrent=16#7FFF,DataPump.PumpCurrent,0)));		Logger.s1:=CONCAT(Logger.s1,';');
Logger.s1:=CONCAT(Logger.s1,WORD_TO_STRING(SEL(DataPump.PumpPower=16#7FFF,DataPump.PumpPower,0)));			Logger.s1:=CONCAT(Logger.s1,';');
Logger.s1:=CONCAT(Logger.s1,WORD_TO_STRING(SEL(DataPump.PumpRPM=16#7FFF,DataPump.PumpRPM,0)));				Logger.s1:=CONCAT(Logger.s1,';');
Logger.s1:=CONCAT(Logger.s1,WORD_TO_STRING(SEL(DataPump.PumpHead=16#7FFF,DataPump.PumpHead,0)));				Logger.s1:=CONCAT(Logger.s1,';');
Logger.s1:=CONCAT(Logger.s1,WORD_TO_STRING(SEL(DataPump.PumpFlow=16#7FFF,DataPump.PumpFlow,0)));				Logger.s1:=CONCAT(Logger.s1,';');
Logger.s1:=CONCAT(Logger.s1,WORD_TO_STRING(SEL(DataPump.PumpLiqTemp=16#7FFF,DataPump.PumpLiqTemp,0)));		Logger.s1:=CONCAT(Logger.s1,';');
Logger.s1:=CONCAT(Logger.s1,DWORD_TO_STRING(SEL(DataPump.PumpOpTime=16#7FFF,DataPump.PumpOpTime,0)));		Logger.s1:=CONCAT(Logger.s1,';');


Logger.s1:=CONCAT(Logger.s1,WORD_TO_STRING(Status_Log));
Logger.s1:=CONCAT(Logger.s1,';');

Logger.s1:=CONCAT(Logger.s1,SEL(DataPump.PumpFault,'0','100'));
Logger.s1:=CONCAT(Logger.s1,';');
Logger.s1:=CONCAT(Logger.s1,SEL(CIR_RUN_REQ,'0','100'));
Logger.s1:=CONCAT(Logger.s1,';');
Logger.s1:=CONCAT(Logger.s1,SEL(CIR_STOP_REQ,'0','100'));

ADDSTRING(ADR(Logger.TData), ADR(Logger.s1), Logger.TLen);
END_ACTION
ACTION CheckFault:
(*** WARNINGS ***)

(* Verify ModBus error	*)
ModbusAlr(IN:=fModbusAlr);

IF ModbusAlr.EVH THEN
	LogEv(EL_Wrn,EO_CIRM,ID,13,SEL(ModBus.MB_MASTER.MB_Error<>0,'0','1'));
	WarningCtr := WarningCtr + 1;
END_IF

IF ModbusAlr.EVL THEN WarningCtr := SEL(WarningCtr=0, WarningCtr-1, 0); END_IF


(*** ALARMS ***)

(* Hardware alarm (physical input *)
AlarmHw(IN:=Pump_AL);

IF AlarmHw.EVH THEN
	LogEv(EL_Alarm,EO_CIRM,ID,3,'CIR_Alarm');
	AlarmCtr := AlarmCtr + 1;
END_IF

IF AlarmHw.EVL THEN
	LogEv(EL_Log,EO_CIRM,ID,4,'CIR_Alarm_Recovered');
	AlarmCtr := SEL(AlarmCtr=0, AlarmCtr-1, 0);
END_IF

(*
(* General alarm (read by Modbus) *)
Alarm(IN:=(DataPump.PumpAlarm[0] <> OldAlarm));

IF Alarm.EVH THEN
	IF DataPump.PumpAlarm[0] = 0 THEN
		LogEv(EL_Log,EO_CIRM,ID,12,'Alarm_Recovered');
		AlarmCtr := SEL(AlarmCtr=0, AlarmCtr-1, 0);
	ELSE
		LogEv(EL_Alarm,EO_CIRM,ID,11,WORD_TO_STRING(DataPump.PumpAlarm[0]));
		AlarmCtr := AlarmCtr + 1;
	END_IF

	OldAlarm := DataPump.PumpAlarm[0];
END_IF


(* Inverter pump error *)
Inverter(IN:=DataPump.PumpFault);

IF Inverter.EVH THEN
	LogEv(EL_Alarm,EO_CIRM,ID,9,'Inverter_Fault');
	AlarmCtr := AlarmCtr + 1;
END_IF

IF Inverter.EVL THEN
	LogEv(EL_Alarm,EO_CIRM,ID,10,'Inverter_Fault_Recovered');
		AlarmCtr := SEL(AlarmCtr=0, AlarmCtr-1, 0);
END_IF

*)
END_ACTION
ACTION Init:
IF NOT InitOK THEN

	Delay.PT_OF := SEL(OffDelay=T#0ms, OffDelay, Plant_CirOffDelay);
	Delay.PT_ON := SEL(OnDelay=T#0ms, OnDelay, Plant_CirOnDelay) + WORD_TO_TIME(1000*ID);

	ReadTmr.PT := WORD_TO_TIME(1000*ID);	(* 1s delay between reads of 2 different double CIRs *)

	Pump_En := 1;
	Refresh_Now := TRUE;

	InitOK := TRUE;

END_IF
END_ACTION
ACTION PumpManager:
(*** Verify Status ***)
IF Pump_AUTO THEN
	IF (Pump_En=1 AND DataPump.PumpStatus=2) OR (Pump_En=0 AND DataPump.PumpStatus=0) THEN fStatusFault := TRUE;
	ELSE fStatusFault := FALSE;
	END_IF
END_IF

fPump_ST(IN:=fStatusFault);

IF fPump_ST.EVH THEN
	LogEv(SEL(Pump_En=1,EL_Alarm,EL_Wrn),EO_CIRM,ID,SEL(Pump_En=1,5,6),'');
	WarningCtr := WarningCtr + 1;
END_IF

IF fPump_ST.EVL THEN WarningCtr := SEL(WarningCtr=0, WarningCtr-1, 0); END_IF

(* Verify if in Auto or Manual mode *)
fCIR_AUTO(IN:=Pump_AUTO);

(* Automatic *)
IF fCIR_AUTO.EVH THEN
	LogEv(EL_Log,EO_CIRM,ID,8,'CIR_Auto');
	WarningCtr := SEL(WarningCtr=0, WarningCtr-1, 0);

	Refresh_Now := TRUE;
END_IF

(* Manual -> Keep switched on *)
IF fCIR_AUTO.EVL THEN
	LogEv(EL_Wrn,EO_CIRM,ID,7,'CIR_Manual');
	WarningCtr := WarningCtr + 1;

	Pump_En := 0;
	Refresh_Now := TRUE;
END_IF

(* Verify if OnOff is changed *)
Ctrl_Run := OnOff;

(* Check switch on or switch off delay *)
Delay(IN:=Ctrl_Run);

IF Pump_AUTO THEN
	(* If priority request *)
	IF CIR_STOP_REQ THEN Pump_En := 1;
	ELSIF CIR_RUN_REQ THEN Pump_En := 0;
	ELSE Pump_En := BOOL_TO_WORD(NOT Delay.OUT);
	END_IF

	(* Set RUN signal (for external objects) *)
	IF AlarmHw.OUT THEN
		Run:=FALSE;
	ELSE
		Run:=SEL(Pump_En=1,TRUE,FALSE);
	END_IF
END_IF

(* Check if a pump enable update (modbus write) is requested *)
fPump_En(IN:=(Pump_En=1));

IF fPump_En.EVH OR fPump_En.EVL THEN
	Refresh_Now := TRUE;
END_IF
END_ACTION
ACTION Stm:
CASE state OF
	WAIT_STATE:	(* Refresh time manager *)
		ReadTmr(IN:=NOT ReadTmr.Q);
		IF ReadTmr.Q OR Refresh_Now  THEN
			state := PUMP_STATUS;
			ReadTmr.PT := T#1m;
			Refresh_Now := FALSE;
		END_IF

	(**** READ CIR PARAMETERS ****)

	PUMP_STATUS:	(* Status and Fault *)
		Modbus.MB_Lock := TRUE;
		Modbus.MB_Query.SlaveAddress := Address;
		Modbus.MB_Query.FunctionCode := 3;
		ModBus.MB_Query.Read_StartAddress := 201;
		ModBus.MB_Query.Read_Quantity := 2;
		ModBus.MB_Start := TRUE;

		state := PUMP_DATA;

	PUMP_DATA:	(* Pump data *)
		IF NOT ModBus.MB_Start AND ModBus.MB_Resp.SlaveAddress=Address  THEN
			IF ModBus.MB_MASTER.bInterfaceError<>0 THEN (*OR ModBus.MB_MASTER.MB_Error<>0 THEN*)
				state := ERROR_STATE;
			ELSE
				DataPump.PumpStatus := ModBus.MB_Resp.Data[0];
				DataPump.PumpFault	:= WORD_TO_BOOL(ModBus.MB_Resp.Data[1]);

				ModBus.MB_Query.Read_StartAddress := 210;
				ModBus.MB_Query.Read_Quantity := 12;
				ModBus.MB_Start := TRUE;

				state := PUMP_ALARMS;
			END_IF
		END_IF

	PUMP_ALARMS: (* Historical alarms *)
		IF NOT ModBus.MB_Start AND ModBus.MB_Resp.SlaveAddress=Address  THEN
			IF ModBus.MB_MASTER.bInterfaceError<>0 THEN (*OR ModBus.MB_MASTER.MB_Error<>0 THEN*)
				state := ERROR_STATE;
			ELSE
				DataPump.PumpBoardTemp 	:= WORD_TO_INT(ModBus.MB_Resp.Data[0]);
				DataPump.PumpVoltage	:= ModBus.MB_Resp.Data[2];
				DataPump.PumpCurrent	:= ModBus.MB_Resp.Data[3];
				DataPump.PumpRPM		:= ModBus.MB_Resp.Data[5];
				DataPump.PumpPower		:= ModBus.MB_Resp.Data[6];
				DataPump.PumpOpTime		:= BUILD_16TO32(ADR(ModBus.MB_Resp.Data[7]));
				DataPump.PumpHead		:= ModBus.MB_Resp.Data[9];
				DataPump.PumpFlow		:= ModBus.MB_Resp.Data[10];
				DataPump.PumpLiqTemp	:= WORD_TO_INT(ModBus.MB_Resp.Data[11]);


				ModBus.MB_Query.Read_StartAddress := 230;
				ModBus.MB_Query.Read_Quantity := 1;(*15;*)
				ModBus.MB_Start := TRUE;

				state := PUMP_END_READ;
			END_IF
		END_IF

	PUMP_END_READ:	(* Read alarms *)
		IF NOT ModBus.MB_Start AND ModBus.MB_Resp.SlaveAddress=Address  THEN
			IF ModBus.MB_MASTER.bInterfaceError<>0 THEN (*OR ModBus.MB_MASTER.MB_Error<>0 THEN*)
				state := ERROR_STATE;
			ELSE
				DataPump.PumpAlarm[0] := ModBus.MB_Resp.Data[0];	(* Read just last (most recent) alarm *)
				(*DataPump.PumpAlarm[1] := ModBus.MB_Resp.Data[1];
				DataPump.PumpAlarm[2] := ModBus.MB_Resp.Data[2];
				DataPump.PumpAlarm[3] := ModBus.MB_Resp.Data[3];
				DataPump.PumpAlarm[4] := ModBus.MB_Resp.Data[4];
				DataPump.PumpAlarm[5] := ModBus.MB_Resp.Data[5];
				DataPump.PumpAlarm[6] := ModBus.MB_Resp.Data[6];
				DataPump.PumpAlarm[7] := ModBus.MB_Resp.Data[7];
				DataPump.PumpAlarm[8] := ModBus.MB_Resp.Data[8];
				DataPump.PumpAlarm[9] := ModBus.MB_Resp.Data[9];
				DataPump.PumpAlarm[10] := ModBus.MB_Resp.Data[10];
				DataPump.PumpAlarm[11] := ModBus.MB_Resp.Data[11];
				DataPump.PumpAlarm[12] := ModBus.MB_Resp.Data[12];
				DataPump.PumpAlarm[13] := ModBus.MB_Resp.Data[13];
				DataPump.PumpAlarm[14] := ModBus.MB_Resp.Data[14];*)

				state := CIR_ON_OFF;

			END_IF
		END_IF

	(**** WRITE ON/OFF REGISTER AND VERIFY RIGHT SETTING ****)
	CIR_ON_OFF:	(* Pump On/off *)

		Modbus.MB_Query.SlaveAddress := Address;
		Modbus.MB_Query.FunctionCode := 6;
		ModBus.MB_Query.Write_StartAddress := 110;
		ModBus.MB_Query.Write_Quantity := 1;
		ModBus.MB_Query.Write_Data[0] := Pump_En;
		ModBus.MB_Start := TRUE;

		state := CIR_END_WRITE;

	CIR_END_WRITE:
		IF NOT ModBus.MB_Start THEN
			IF ModBus.MB_MASTER.bInterfaceError<>0 THEN (*OR ModBus.MB_MASTER.MB_Error<>0 THEN*)
				state := ERROR_STATE;
			ELSE
				IF fModbusAlr THEN fModbusAlr := FALSE; END_IF

				ModBus.MB_Lock := FALSE;
				retryErr := 0;
				retry := 0;
				state := WAIT_STATE;
			END_IF
		END_IF


	(**** CHECK MODBUS ERROR ****)
	ERROR_STATE: 	(* Release MODBUS *)
			MODBUS.MB_Lock:=FALSE;

			(* Retries *)
			retry:=retry+1;
			IF retry>3 THEN
				retry:=0;

				(* Verify if slave is dead *)
				IF retryErr < retryErrMaX THEN
					retryErr := retryErr + 1;
				ELSE
					fModbusAlr := TRUE;
				END_IF

				Refresh_Now := FALSE;
			END_IF

			state:=WAIT_STATE;
END_CASE

(* Controllo Time Out Ciclo ModBus *)

TimeOutModBus(In:=state<>0,PT:=t#2s);
IF TimeOutModBus.Q THEN State:=0; END_IF
END_ACTION

(* POU Plant_Objects/obj_MODBUS_CIR_DOPPIO_new, ST *)
FUNCTION_BLOCK obj_MODBUS_CIR_DOPPIO_new
VAR CONSTANT
	WAIT_STATE		:	BYTE := 0;
	PUMP1_STATUS	:	BYTE := 1;
	PUMP1_DATA		:	BYTE := 2;
	PUMP1_ALARMS	:	BYTE := 3;
	PUMP1_END_READ	:	BYTE := 4;
	PUMP2_STATUS	:	BYTE := 5;
	PUMP2_DATA		:	BYTE := 6;
	PUMP2_ALARMS	:	BYTE := 7;
	PUMP2_END_READ	:	BYTE := 8;
	CIR_ON_OFF1		:	BYTE := 90;
	CIR_ON_OFF2		:	BYTE := 91;
	CIR_ON_OFF_CHECK:	BYTE := 92;
	CIR_END_WRITE	:	BYTE := 93;
	ERROR_STATE		:	BYTE := 100;

END_VAR
VAR_INPUT
	ID		:	BYTE;
	Address1:	BYTE;		(* Pump 1 Modbus address *)
	Address2:	BYTE;		(* Pump 2 Modbus address *)

	(* Physical inputs (Force) *)
	CIR_RUN_REQ		: BOOL; (* External run request (no heat or cold requested) *)
	CIR_STOP_REQ	: BOOL; (* External stop request (has priority over RUN signals!) *)

	(* Physical inputs (Feedback) *)
	PumpA_AL		: BOOL; (* Alarm input signal *)
	PumpB_AL		: BOOL;
	PumpA_AUTO		: BOOL;	(* Automatic/Manual input *)
	PumpB_AUTO		: BOOL;

	(* Controls *)
	OnOff		: 	BOOL;	(* On/Off from chrono *)
	Mode		:	BYTE;	(* Working mode: 0-Both pumps works simultaneously, 1-Alternate every 24h, 2-Master/Backup *)
	InitOK		:	BOOL;

	(* Timings *)
	OnDelay		:	TIME;	(* Switch on delay *)
	OffDelay	:	TIME;	(* Switch off delay *)

	(* Modbus *)
	Refresh_Now	:	BOOL;	(* Start immediately modbus state machine *)
	retryErrMax	:	BYTE := 15;
END_VAR
VAR_IN_OUT
	ModBus		:	obj_MODBUS;
END_VAR
VAR_OUTPUT
	Ctrl_Run	:	BOOL;		(* Logical status of the device: 0: Not running (switched off), 1: running *)
	Run			:	BOOL;		(* Real status *)

	Status_Log	:	WORD;
	Status_Vis	:	DWORD;
END_VAR
VAR
	Status		:	BOOL;
	Pump_En		:	ARRAY [1..2] OF WORD;		(* Pumps enable *)

	ChangeTmr	: 	TON := (PT:=T#24h);			(* Timer that counts change time when in alternate mode *)
	ActivePump	: 	BYTE := 1;						(* Actual active pump *)
	NewActivePump	: BYTE := 1;

	(* Filters *)
	fPump_ST	: 	ARRAY [1..2] OF FLT_TAP := (INITEV:=FALSE);
	fPump_En	:	ARRAY [1..2] OF FLT_EVENT;
	fCIR_AUTO	:	ARRAY [1..2] OF FLT_TAP;
	fStatusFault:	ARRAY [1..2] OF BOOL;
	fBackup		:	FLT_EVENT := (INITEV:=FALSE);

	(* Timer manage switch on/off delay *)
	Delay		: 	TONOF;

	(* CIR data structure *)
	DataPump1	:	typ_MODBUS_CIR;
	DataPump2	:	typ_MODBUS_CIR;

	(* Modbus variables *)
	state		:	BYTE;
	retry		:	BYTE;
	retryErr	:	BYTE;
	ReadTmr		:	TON := (PT:=T#5s);
	fModbusAlr	: 	BOOL;

	(* Alarm and Warning counters *)
	AlarmCtr	:	BYTE;
	WarningCtr	:	BYTE;

	(* Filers on alarms and faults *)
	AlarmHw		:	ARRAY [1..2] OF FLT_TAP := (INITEV:=FALSE);
	Alarm		:	ARRAY [1..2] OF FLT_EVENT := (INITEV:=FALSE);
	Inverter	:	ARRAY [1..2] OF FLT_EVENT := (INITEV:=FALSE);
	ModbusAlr	:	FLT_EVENT := (INITEV:=FALSE);

	OldAlarmPump1	:	WORD;
	OldAlarmPump2	:	WORD;

	TimeOutModBus: TON;
END_VAR
Init();

(* Check alarm and warning for both pumps *)
CheckFault();

PumpManager();

(* State machine to read pump parameters *)
Stm();

IF AlarmCtr>0 THEN
	Status_Log := 2;
	Status_Vis := COLOR_RED;
ELSIF WarningCtr>0 THEN
	Status_Log := 1;
	Status_Vis := COLOR_YELLOW;
ELSE
	Status_Log := 0;
	Status_Vis := COLOR_GREEN;
END_IF

(* Update error lamp status *)
Lamp.UpdateStatus(obj_Status := Status_Log);
END_FUNCTION_BLOCK
ACTION AddLogData:
Logger.s1:=INSERT('&CIRDM=',BYTE_TO_STRING(ID),6);
IF ID<10 THEN Logger.s1:=INSERT(Logger.s1,'0',6); END_IF

Logger.s1:=CONCAT(Logger.s1,WORD_TO_STRING(Mode));						Logger.s1:=CONCAT(Logger.s1,';');
(* PUMP 1 *)
(* NB If value equals 0x7FFF (32767) this means that it is not available -->> Change it to 0 *)
Logger.s1:=CONCAT(Logger.s1,WORD_TO_STRING(DataPump1.PumpStatus));											Logger.s1:=CONCAT(Logger.s1,';');
Logger.s1:=CONCAT(Logger.s1,INT_TO_STRING(SEL(DataPump1.PumpBoardTemp=16#7FFF,DataPump1.PumpBoardTemp,0)));	Logger.s1:=CONCAT(Logger.s1,';');
Logger.s1:=CONCAT(Logger.s1,WORD_TO_STRING(SEL(DataPump1.PumpVoltage=16#7FFF,DataPump1.PumpVoltage,0)));		Logger.s1:=CONCAT(Logger.s1,';');
Logger.s1:=CONCAT(Logger.s1,WORD_TO_STRING(SEL(DataPump1.PumpCurrent=16#7FFF,DataPump1.PumpCurrent,0)));		Logger.s1:=CONCAT(Logger.s1,';');
Logger.s1:=CONCAT(Logger.s1,WORD_TO_STRING(SEL(DataPump1.PumpPower=16#7FFF,DataPump1.PumpPower,0)));			Logger.s1:=CONCAT(Logger.s1,';');
Logger.s1:=CONCAT(Logger.s1,WORD_TO_STRING(SEL(DataPump1.PumpRPM=16#7FFF,DataPump1.PumpRPM,0)));				Logger.s1:=CONCAT(Logger.s1,';');
Logger.s1:=CONCAT(Logger.s1,WORD_TO_STRING(SEL(DataPump1.PumpHead=16#7FFF,DataPump1.PumpHead,0)));				Logger.s1:=CONCAT(Logger.s1,';');
Logger.s1:=CONCAT(Logger.s1,WORD_TO_STRING(SEL(DataPump1.PumpFlow=16#7FFF,DataPump1.PumpFlow,0)));				Logger.s1:=CONCAT(Logger.s1,';');
Logger.s1:=CONCAT(Logger.s1,WORD_TO_STRING(SEL(DataPump1.PumpLiqTemp=16#7FFF,DataPump1.PumpLiqTemp,0)));		Logger.s1:=CONCAT(Logger.s1,';');
Logger.s1:=CONCAT(Logger.s1,DWORD_TO_STRING(SEL(DataPump1.PumpOpTime=16#7FFF,DataPump1.PumpOpTime,0)));		Logger.s1:=CONCAT(Logger.s1,';');


(* PUMP 2 *)
Logger.s1:=CONCAT(Logger.s1,WORD_TO_STRING(DataPump2.PumpStatus));											Logger.s1:=CONCAT(Logger.s1,';');
Logger.s1:=CONCAT(Logger.s1,INT_TO_STRING(SEL(DataPump2.PumpBoardTemp=16#7FFF,DataPump2.PumpBoardTemp,0)));	Logger.s1:=CONCAT(Logger.s1,';');
Logger.s1:=CONCAT(Logger.s1,WORD_TO_STRING(SEL(DataPump2.PumpVoltage=16#7FFF,DataPump2.PumpVoltage,0)));		Logger.s1:=CONCAT(Logger.s1,';');
Logger.s1:=CONCAT(Logger.s1,WORD_TO_STRING(SEL(DataPump2.PumpCurrent=16#7FFF,DataPump2.PumpCurrent,0)));		Logger.s1:=CONCAT(Logger.s1,';');
Logger.s1:=CONCAT(Logger.s1,WORD_TO_STRING(SEL(DataPump2.PumpPower=16#7FFF,DataPump2.PumpPower,0)));			Logger.s1:=CONCAT(Logger.s1,';');
Logger.s1:=CONCAT(Logger.s1,WORD_TO_STRING(SEL(DataPump2.PumpRPM=16#7FFF,DataPump2.PumpRPM,0)));				Logger.s1:=CONCAT(Logger.s1,';');
Logger.s1:=CONCAT(Logger.s1,WORD_TO_STRING(SEL(DataPump2.PumpHead=16#7FFF,DataPump2.PumpHead,0)));				Logger.s1:=CONCAT(Logger.s1,';');
Logger.s1:=CONCAT(Logger.s1,WORD_TO_STRING(SEL(DataPump2.PumpFlow=16#7FFF,DataPump2.PumpFlow,0)));				Logger.s1:=CONCAT(Logger.s1,';');
Logger.s1:=CONCAT(Logger.s1,WORD_TO_STRING(SEL(DataPump2.PumpLiqTemp=16#7FFF,DataPump2.PumpLiqTemp,0)));		Logger.s1:=CONCAT(Logger.s1,';');
Logger.s1:=CONCAT(Logger.s1,DWORD_TO_STRING(SEL(DataPump2.PumpOpTime=16#7FFF,DataPump2.PumpOpTime,0)));		Logger.s1:=CONCAT(Logger.s1,';');

Logger.s1:=CONCAT(Logger.s1,WORD_TO_STRING(Status_Log));
Logger.s1:=CONCAT(Logger.s1,';');

Logger.s1:=CONCAT(Logger.s1,SEL(DataPump1.PumpFault,'0','100'));
Logger.s1:=CONCAT(Logger.s1,';');
Logger.s1:=CONCAT(Logger.s1,SEL(DataPump2.PumpFault,'0','100'));
Logger.s1:=CONCAT(Logger.s1,';');
Logger.s1:=CONCAT(Logger.s1,SEL(CIR_RUN_REQ,'0','100'));
Logger.s1:=CONCAT(Logger.s1,';');
Logger.s1:=CONCAT(Logger.s1,SEL(CIR_STOP_REQ,'0','100'));






ADDSTRING(ADR(Logger.TData), ADR(Logger.s1), Logger.TLen);
END_ACTION
ACTION CheckFault:
(*** WARNINGS ***)

(* Verify ModBus error	*)
ModbusAlr(IN:=fModbusAlr);

IF ModbusAlr.EVH THEN
	LogEv(EL_Alarm,EO_CIRDM,ID,13,SEL(ModBus.MB_MASTER.MB_Error<>0,'0','1'));
	WarningCtr := WarningCtr + 1;
END_IF

IF ModbusAlr.EVL THEN
	LogEv(EL_Log,EO_CIRDM,ID,14,'');
	WarningCtr := SEL(WarningCtr=0, WarningCtr-1, 0);
END_IF


(*** ALARMS ***)

(**** PUMP 1 ****)

(* Hardware alarm (physical input *)
AlarmHw[1](IN:=PumpA_AL);

IF AlarmHw[1].EVH THEN
	LogEv(EL_Alarm,EO_CIRDM,ID,3,'1');
	AlarmCtr := AlarmCtr + 1;
END_IF

IF AlarmHw[1].EVL THEN
	LogEv(EL_Log,EO_CIRDM,ID,4,'1');
	AlarmCtr := SEL(AlarmCtr=0, AlarmCtr-1, 0);
END_IF

(*
(* General alarm (read by Modbus) *)
Alarm[1](IN:=(DataPump1.PumpAlarm[0] <> OldAlarmPump1));

IF Alarm[1].EVH THEN
	IF DataPump1.PumpAlarm[1] = 0 THEN
		LogEv(EL_Alarm,EO_CIRDM,ID,11,'1');
		AlarmCtr := SEL(AlarmCtr=0, AlarmCtr-1, 0);
	ELSE
		LogEv(EL_Alarm,EO_CIRDM,ID,12,WORD_TO_STRING(DataPump1.PumpAlarm[1]));
		AlarmCtr := AlarmCtr + 1;
	END_IF

	OldAlarmPump1 := DataPump1.PumpAlarm[1];
END_IF

(* Inverter pump error *)
Inverter[1](IN:=DataPump1.PumpFault);

IF Inverter[1].EVH THEN
	LogEv(EL_Alarm,EO_CIRDM,ID,9,'1');
	AlarmCtr := AlarmCtr + 1;
END_IF

IF Inverter[1].EVL THEN
	LogEv(EL_Alarm,EO_CIRDM,ID,10,'1');
	AlarmCtr := SEL(AlarmCtr=0, AlarmCtr-1, 0);
END_IF
*)

(**** PUMP 2 ****)

(* Hardware alarm (physical input *)
AlarmHw[2](IN:=PumpB_AL);

IF AlarmHw[2].EVH THEN
	LogEv(EL_Alarm,EO_CIRDM,ID,3,'2');
	AlarmCtr := AlarmCtr + 1;
END_IF

IF AlarmHw[2].EVL THEN
	LogEv(EL_Log,EO_CIRDM,ID,4,'2');
	AlarmCtr := SEL(AlarmCtr=0, AlarmCtr-1, 0);
END_IF

(*
(* General alarm (read by Modbus) *)
Alarm[2](IN:=(DataPump2.PumpAlarm[0] <> OldAlarmPump2));

IF Alarm[2].EVH THEN
	IF DataPump2.PumpAlarm[0] = 0 THEN
		LogEv(EL_Log,EO_CIRDM,ID,11,'2');
		AlarmCtr := SEL(AlarmCtr=0, AlarmCtr-1, 0);
	ELSE
		LogEv(EL_Alarm,EO_CIRDM,ID,12,WORD_TO_STRING(DataPump2.PumpAlarm[0]));
		AlarmCtr := AlarmCtr + 1;
	END_IF

	OldAlarmPump2 := DataPump2.PumpAlarm[0];
END_IF

(* Inverter pump error *)
Inverter[2](IN:=DataPump2.PumpFault);

IF Inverter[2].EVH THEN
	LogEv(EL_Alarm,EO_CIRDM,ID,9,'2');
	AlarmCtr := AlarmCtr + 1;
END_IF

IF Inverter[2].EVL THEN
	LogEv(EL_Log,EO_CIRDM,ID,10,'2');
	AlarmCtr := SEL(AlarmCtr=0, AlarmCtr-1, 0);
END_IF
*)
END_ACTION
ACTION Init:
IF NOT InitOK THEN

	Delay.PT_OF := SEL(OffDelay=T#0s, OffDelay, Plant_CirOffDelay);
	Delay.PT_ON := SEL(OnDelay=T#0s, OnDelay, Plant_CirOnDelay) + WORD_TO_TIME(1000*ID);

	ReadTmr.PT := WORD_TO_TIME(2000*ID);	(* 1s delay between reads of 2 different double CIRs *)

	Pump_En[1] := 1;
	Pump_En[2] := 1;

	Refresh_Now := TRUE;
	InitOK := TRUE;

END_IF
END_ACTION
ACTION PumpManager:
(*** Verify Status ***)
IF PumpA_AUTO THEN
	IF (Pump_En[1]=1 AND DataPump1.PumpStatus=2) OR (Pump_En[1]=0 AND DataPump1.PumpStatus=0) THEN fStatusFault[1] := TRUE;
	ELSE fStatusFault[1] := FALSE;
	END_IF
END_IF

IF PumpB_AUTO THEN
	IF (Pump_En[2]=1 AND DataPump2.PumpStatus=2) OR (Pump_En[2]=0 AND DataPump2.PumpStatus=0) THEN fStatusFault[2] := TRUE;
	ELSE fStatusFault[2] := FALSE;
	END_IF
END_IF

fPump_ST[1](IN:=fStatusFault[1]);
fPump_ST[2](IN:=fStatusFault[2]);

IF fPump_ST[1].EVH THEN
	LogEv(SEL(Pump_En[1]=1,EL_Alarm,EL_Wrn),EO_CIRDM,ID,SEL(Pump_En[1]=1,5,6),'1');
	WarningCtr := WarningCtr + 1;
END_IF

IF fPump_ST[1].EVL THEN WarningCtr := SEL(WarningCtr=0, WarningCtr-1, 0); END_IF

IF fPump_ST[2].EVH THEN
	LogEv(SEL(Pump_En[2]=1,EL_Alarm,EL_Wrn),EO_CIRDM,ID,SEL(Pump_En[2]=1,5,6),'2');
	WarningCtr := WarningCtr + 1;
END_IF

IF fPump_ST[2].EVL THEN WarningCtr := SEL(WarningCtr=0, WarningCtr-1, 0); END_IF


(* Verify if in Auto or Manual mode *)
fCIR_AUTO[1](IN:=PumpA_AUTO);
fCIR_AUTO[2](IN:=PumpB_AUTO);

(*** Pump A ***)
IF fCIR_AUTO[1].EVH THEN
	LogEv(EL_Log,EO_CIRDM,ID,8,'1');
	WarningCtr := SEL(WarningCtr=0, WarningCtr-1, 0);

	IF ActivePump=2 THEN Pump_En[1] := 1; END_IF
	Refresh_Now := TRUE;
END_IF

(* Manual -> Keep switched on *)
IF fCIR_AUTO[1].EVL THEN
	LogEv(EL_Wrn,EO_CIRDM,ID,7,'1');
	WarningCtr := WarningCtr + 1;

	(* Switch on pump A *)
	Pump_En[1] := 0;
(*	Run := TRUE;
	Ctrl_Run := TRUE;*)
	Refresh_Now := TRUE;
END_IF

(*** Pump B ***)
IF fCIR_AUTO[2].EVH THEN
	LogEv(EL_Log,EO_CIRDM,ID,8,'2');
	WarningCtr := SEL(WarningCtr=0, WarningCtr-1, 0);

	IF ActivePump=1 THEN Pump_En[2] := 1; END_IF
	Refresh_Now := TRUE;
END_IF

(* Manual -> Keep switched on *)
IF fCIR_AUTO[2].EVL THEN
	LogEv(EL_Wrn,EO_CIRDM,ID,7,'2');
	WarningCtr := WarningCtr + 1;

	(* Switch on pump B *)
	Pump_En[2] := 0;
(*	Ctrl_Run := TRUE;
	Run := TRUE;*)
	Refresh_Now := TRUE;
END_IF

IF PumpA_AUTO AND PumpB_AUTO THEN
	(* Verify if OnOff is changed *)
	Ctrl_Run := OnOff;
END_IF

(* Check switch on or switch off delay *)
Delay(IN:=Ctrl_Run);

(* If working mode is Alternate, count change time *)
IF Mode=1 THEN

	ChangeTmr(IN:=NOT ChangeTmr.Q);

	IF ChangeTmr.Q THEN

		NewActivePump := SEL(ActivePump=1,1,2);

		(* If no alarm on other pump, keep going with the switch *)
		IF NOT AlarmHw[NewActivePump].OUT THEN ActivePump := NewActivePump;
		ELSE LogEv(EL_Wrn,EO_CIRDM,ID,15,'');		(* Pump not switched because of other pump's failure *)
		END_IF

		(* Switch off old active pump *)
		IF ActivePump=1 THEN Pump_En[2] := 1;
		ELSE Pump_En[1] := 1;
		END_IF

		(* Write new parameters (also if not changed) *)
		Refresh_Now := TRUE;
		ChangeTmr.PT:=T#24h;
	END_IF
END_IF


(* Set output according to actual function mode *)
CASE Mode OF

	0:	(*** Simultaneous pumps working ***)
		IF PumpA_AUTO THEN

			IF CIR_STOP_REQ THEN Pump_En[1] := 1;
			ELSIF CIR_RUN_REQ THEN Pump_En[1] := 0;
			ELSE Pump_En[1] := BOOL_TO_WORD(NOT Delay.OUT);
			END_IF

			(* Set RUN signal (for external objects) *)
			IF AlarmCtr>0 THEN (*OR fPump_ST[1].OUT OR fPump_ST[2].OUT THEN*)
				Run:=FALSE;
			ELSE
				Run:=SEL(Pump_En[1]=1,TRUE,FALSE);
			END_IF
		END_IF

		IF PumpB_AUTO THEN

			IF CIR_STOP_REQ THEN Pump_En[2] := 1;
			ELSIF CIR_RUN_REQ THEN Pump_En[2] := 0;
			ELSE Pump_En[2] := BOOL_TO_WORD(NOT Delay.OUT);
			END_IF

			(* Set RUN signal (for external objects) *)
			IF AlarmCtr>0 THEN (*OR fPump_ST[1].OUT OR fPump_ST[2].OUT THEN*)
				Run:=FALSE;
			ELSE
				Run:=SEL(Pump_En[2]=1,FALSE,TRUE);
			END_IF
		END_IF


	1,2:  (*** Alternate working and Master/backup mode ***)
		IF fCIR_AUTO[ActivePump].IN THEN
			(* If priority request *)
			IF CIR_STOP_REQ THEN Pump_En[ActivePump] := 1;
			ELSIF CIR_RUN_REQ THEN Pump_En[ActivePump] := 0;
			ELSE Pump_En[ActivePump] := BOOL_TO_WORD(NOT Delay.OUT);
			END_IF

			fBackup(IN:=(AlarmHw[ActivePump].OUT));

			IF fBackup.EVH THEN
				ActivePump := SEL(ActivePump=1,1,2);
				LogEv(EL_Wrn,EO_CIRD,ID,16,'');	(* Pump switched because of current pump failure *)

				(* Switch off old active pump *)
				IF ActivePump=1 THEN Pump_En[2] := 1;
				ELSE Pump_En[1] := 1;
				END_IF
			END_IF


			(* Set RUN signal (for external objects) *)
			IF AlarmCtr>0 THEN (*OR fPump_ST[ActivePump].OUT THEN*)
				Run:=FALSE;
			ELSE
				IF (ActivePump=1 AND PumpB_AUTO) OR (ActivePump=2 AND PumpA_AUTO) THEN
					Run:=SEL(Pump_En[ActivePump]=1,TRUE,FALSE);
				END_IF
			END_IF

		END_IF

END_CASE

(* Check if a pump enable update (modbus write) is requested *)
fPump_En[1](IN:=(Pump_En[1]=1));
fPump_En[2](IN:=(Pump_En[2]=1));

IF fPump_En[1].EVH OR fPump_En[1].EVL THEN
	Refresh_Now := TRUE;
END_IF

IF fPump_En[2].EVH OR fPump_En[2].EVL THEN
	Refresh_Now := TRUE;
END_IF
END_ACTION
ACTION Stm:
CASE state OF
	WAIT_STATE:	(* Refresh time manager *)
		ReadTmr(IN:=NOT ReadTmr.Q);
		IF ReadTmr.Q OR Refresh_Now THEN
			state := PUMP1_STATUS;
			ReadTmr.PT := T#1m;

		END_IF

	(**** READ CIR PARAMETERS ****)

	(**** PUMP 1 ****)
	PUMP1_STATUS:	(* Status and Fault *)
		IF NOT Modbus.MB_Lock THEN
			Modbus.MB_Lock := TRUE;
	
			Modbus.MB_Query.SlaveAddress := Address1;
			Modbus.MB_Query.FunctionCode := 3;
			ModBus.MB_Query.Read_StartAddress := 201;
			ModBus.MB_Query.Read_Quantity := 2;
			ModBus.MB_Start := TRUE;

			state := PUMP1_DATA;
		END_IF

	PUMP1_DATA:	(* Pump data *)
		IF NOT ModBus.MB_Start AND ModBus.MB_Resp.SlaveAddress=Address1 THEN
			IF ModBus.MB_MASTER.bInterfaceError<>0 THEN (*OR ModBus.MB_MASTER.MB_Error<>0 THEN*)
				state := ERROR_STATE;
			ELSE
				DataPump1.PumpStatus := ModBus.MB_Resp.Data[0];
				DataPump1.PumpFault	:= WORD_TO_BOOL(ModBus.MB_Resp.Data[1]);

				Modbus.MB_Query.SlaveAddress := Address1;
				Modbus.MB_Query.FunctionCode := 3;
				ModBus.MB_Query.Read_StartAddress := 210;
				ModBus.MB_Query.Read_Quantity := 12;
				ModBus.MB_Start := TRUE;

				state := PUMP1_ALARMS;
			END_IF
		END_IF

	PUMP1_ALARMS: (* Historical alarms *)
		IF NOT ModBus.MB_Start AND ModBus.MB_Resp.SlaveAddress=Address1 THEN
			IF ModBus.MB_MASTER.bInterfaceError<>0 THEN (*OR ModBus.MB_MASTER.MB_Error<>0 THEN*)
				state := ERROR_STATE;
			ELSE
				DataPump1.PumpBoardTemp := WORD_TO_INT(ModBus.MB_Resp.Data[0]);
				DataPump1.PumpVoltage	:= ModBus.MB_Resp.Data[2];
				DataPump1.PumpCurrent	:= ModBus.MB_Resp.Data[3];
				DataPump1.PumpRPM		:= ModBus.MB_Resp.Data[5];
				DataPump1.PumpPower		:= ModBus.MB_Resp.Data[6];
				DataPump1.PumpOpTime	:= BUILD_16TO32(ADR(ModBus.MB_Resp.Data[7]));
				DataPump1.PumpHead		:= ModBus.MB_Resp.Data[9];
				DataPump1.PumpFlow		:= ModBus.MB_Resp.Data[10];
				DataPump1.PumpLiqTemp	:= WORD_TO_INT(ModBus.MB_Resp.Data[11]);

				Modbus.MB_Query.SlaveAddress := Address1;
				Modbus.MB_Query.FunctionCode := 3;
				ModBus.MB_Query.Read_StartAddress := 230;
				ModBus.MB_Query.Read_Quantity := 1;(*15;*)
				ModBus.MB_Start := TRUE;

				state := PUMP1_END_READ;
			END_IF
		END_IF

	PUMP1_END_READ:	(* Read alarms *)
		IF NOT ModBus.MB_Start AND ModBus.MB_Resp.SlaveAddress=Address1 THEN
			IF ModBus.MB_MASTER.bInterfaceError<>0 THEN (*OR ModBus.MB_MASTER.MB_Error<>0 THEN*)
				state := ERROR_STATE;
			ELSE
				DataPump1.PumpAlarm[0] := ModBus.MB_Resp.Data[0];
				(*DataPump1.PumpAlarm[1] := ModBus.MB_Resp.Data[1];
				DataPump1.PumpAlarm[2] := ModBus.MB_Resp.Data[2];
				DataPump1.PumpAlarm[3] := ModBus.MB_Resp.Data[3];
				DataPump1.PumpAlarm[4] := ModBus.MB_Resp.Data[4];
				DataPump1.PumpAlarm[5] := ModBus.MB_Resp.Data[5];
				DataPump1.PumpAlarm[6] := ModBus.MB_Resp.Data[6];
				DataPump1.PumpAlarm[7] := ModBus.MB_Resp.Data[7];
				DataPump1.PumpAlarm[8] := ModBus.MB_Resp.Data[8];
				DataPump1.PumpAlarm[9] := ModBus.MB_Resp.Data[9];
				DataPump1.PumpAlarm[10] := ModBus.MB_Resp.Data[10];
				DataPump1.PumpAlarm[11] := ModBus.MB_Resp.Data[11];
				DataPump1.PumpAlarm[12] := ModBus.MB_Resp.Data[12];
				DataPump1.PumpAlarm[13] := ModBus.MB_Resp.Data[13];
				DataPump1.PumpAlarm[14] := ModBus.MB_Resp.Data[14];*)

				state := PUMP2_STATUS;
			END_IF
		END_IF

	(**** PUMP 2 ****)
	PUMP2_STATUS:	(* Status and Fault *)

		Modbus.MB_Query.SlaveAddress := Address2;
		Modbus.MB_Query.FunctionCode := 3;
		ModBus.MB_Query.Read_StartAddress := 201;
		ModBus.MB_Query.Read_Quantity := 2;
		ModBus.MB_Start := TRUE;

		state := PUMP2_DATA;

	PUMP2_DATA:	(* Pump data *)
		IF NOT ModBus.MB_Start AND ModBus.MB_Resp.SlaveAddress=Address2 THEN
			IF ModBus.MB_MASTER.bInterfaceError<>0 THEN (*OR ModBus.MB_MASTER.MB_Error<>0 THEN*)
				state := ERROR_STATE;
			ELSE
				DataPump2.PumpStatus := ModBus.MB_Resp.Data[0];
				DataPump2.PumpFault	:= WORD_TO_BOOL(ModBus.MB_Resp.Data[1]);

				Modbus.MB_Query.SlaveAddress := Address2;
				Modbus.MB_Query.FunctionCode := 3;
				ModBus.MB_Query.Read_StartAddress := 210;
				ModBus.MB_Query.Read_Quantity := 12;
				ModBus.MB_Start := TRUE;

				state := PUMP2_ALARMS;
			END_IF
		END_IF

	PUMP2_ALARMS:
		IF NOT ModBus.MB_Start AND ModBus.MB_Resp.SlaveAddress=Address2 THEN
			IF ModBus.MB_MASTER.bInterfaceError<>0 THEN (*OR ModBus.MB_MASTER.MB_Error<>0 THEN*)
				state := ERROR_STATE;
			ELSE
				DataPump2.PumpBoardTemp := WORD_TO_INT(ModBus.MB_Resp.Data[0]);
				DataPump2.PumpVoltage	:= ModBus.MB_Resp.Data[2];
				DataPump2.PumpCurrent	:= ModBus.MB_Resp.Data[3];
				DataPump2.PumpRPM		:= ModBus.MB_Resp.Data[5];
				DataPump2.PumpPower		:= ModBus.MB_Resp.Data[6];
				DataPump2.PumpOpTime	:= BUILD_16TO32(ADR(ModBus.MB_Resp.Data[7]));
				DataPump2.PumpHead		:= ModBus.MB_Resp.Data[9];
				DataPump2.PumpFlow		:= ModBus.MB_Resp.Data[10];
				DataPump2.PumpLiqTemp	:= WORD_TO_INT(ModBus.MB_Resp.Data[11]);

				Modbus.MB_Query.SlaveAddress := Address2;
				Modbus.MB_Query.FunctionCode := 3;
				ModBus.MB_Query.Read_StartAddress := 230;
				ModBus.MB_Query.Read_Quantity := 15;
				ModBus.MB_Start := TRUE;

				state := PUMP2_END_READ;
			END_IF
		END_IF

	PUMP2_END_READ:
		IF NOT ModBus.MB_Start AND ModBus.MB_Resp.SlaveAddress=Address2 THEN
			IF ModBus.MB_MASTER.bInterfaceError<>0 THEN (*OR ModBus.MB_MASTER.MB_Error<>0 THEN*)
				state := ERROR_STATE;
			ELSE
				DataPump2.PumpAlarm[0] := ModBus.MB_Resp.Data[0];
				DataPump2.PumpAlarm[1] := ModBus.MB_Resp.Data[1];
				DataPump2.PumpAlarm[2] := ModBus.MB_Resp.Data[2];
				DataPump2.PumpAlarm[3] := ModBus.MB_Resp.Data[3];
				DataPump2.PumpAlarm[4] := ModBus.MB_Resp.Data[4];
				DataPump2.PumpAlarm[5] := ModBus.MB_Resp.Data[5];
				DataPump2.PumpAlarm[6] := ModBus.MB_Resp.Data[6];
				DataPump2.PumpAlarm[7] := ModBus.MB_Resp.Data[7];
				DataPump2.PumpAlarm[8] := ModBus.MB_Resp.Data[8];
				DataPump2.PumpAlarm[9] := ModBus.MB_Resp.Data[9];
				DataPump2.PumpAlarm[10] := ModBus.MB_Resp.Data[10];
				DataPump2.PumpAlarm[11] := ModBus.MB_Resp.Data[11];
				DataPump2.PumpAlarm[12] := ModBus.MB_Resp.Data[12];
				DataPump2.PumpAlarm[13] := ModBus.MB_Resp.Data[13];
				DataPump2.PumpAlarm[14] := ModBus.MB_Resp.Data[14];

				Modbus.MB_Query.SlaveAddress := Address1;
				Modbus.MB_Query.FunctionCode := 6;
				ModBus.MB_Query.Write_StartAddress := 110;
				ModBus.MB_Query.Write_Quantity := 1;
				ModBus.MB_Query.Write_Data[0] := Pump_En[1];
				ModBus.MB_Start := TRUE;

				state := CIR_ON_OFF1;
			END_IF
		END_IF

	(**** WRITE ON/OFF REGISTER AND VERIFY RIGHT SETTING ****)

	CIR_ON_OFF1:	(* Pump A On/off *)
		IF NOT ModBus.MB_Start THEN
			IF ModBus.MB_MASTER.bInterfaceError<>0 THEN (*OR ModBus.MB_MASTER.MB_Error<>0 THEN*)
				state := ERROR_STATE;
			ELSE
				Modbus.MB_Query.SlaveAddress := Address2;
				Modbus.MB_Query.FunctionCode := 6;
				ModBus.MB_Query.Write_StartAddress := 110;
				ModBus.MB_Query.Write_Quantity := 1;
				ModBus.MB_Query.Write_Data[0] := Pump_En[2];
				ModBus.MB_Start := TRUE;

				state := CIR_ON_OFF2;
			END_IF
		END_IF

	CIR_ON_OFF2:

		IF NOT ModBus.MB_Start THEN
			IF ModBus.MB_MASTER.bInterfaceError<>0 THEN (*OR ModBus.MB_MASTER.MB_Error<>0 THEN*)
				state := ERROR_STATE;
			ELSE
				IF fModbusAlr THEN fModbusAlr := FALSE; END_IF

				Refresh_Now := FALSE;
				ModBus.MB_Lock := FALSE;
				retry := 0;
				retryErr := 0;
				state := WAIT_STATE;
			END_IF
		END_IF

	(**** CHECK MODBUS ERROR ****)
	ERROR_STATE: 	(* Release MODBUS *)
			MODBUS.MB_Lock:=FALSE;

			(* Retries *)
			retry:=retry+1;
			IF retry>3 THEN
				retry:=0;
				(* Verify if slave is dead *)
				IF retryErr < retryErrMaX THEN
					retryErr := retryErr + 1;
				ELSE
					fModbusAlr := TRUE;
				END_IF

				Refresh_Now := FALSE;
			END_IF

			state:=WAIT_STATE;
END_CASE

(* Controllo Time Out Ciclo ModBus *)

TimeOutModBus(In:=state<>0,PT:=t#2s);
IF TimeOutModBus.Q THEN State:=0; END_IF
END_ACTION

(* POU Plant_Objects/obj_MODBUS_TCP, ST *)
FUNCTION_BLOCK obj_MODBUS_TCP
(* === MODBUS-TCP PROTOCOL INTERFACE ===
   v1.0[10/06/15] - Create
*)
VAR CONSTANT
	VARS_Max	: BYTE := 32;
END_VAR
VAR_INPUT
	(* Settings *)
	ID			: BYTE;
	IP			: STRING;
	PORT		: WORD:=502;
	(* Interface *)
	MB_MASTER	: ETHERNET_MODBUSMASTER_TCP;
	MB_READBUF	: ARRAY [0..128] OF WORD;
	MB_WRITEBUF : ARRAY [0..128] OF WORD;
	MB_Start	: BOOL;
	MB_Lock		: BOOL;
	(* Variables management *)
	VARS_En		: BOOL;
	VARS		: ARRAY [0..VARS_Max] OF typ_MODBUS_VAR;
	VARS_Check	: BOOL;
	VARS_Alarm	: BOOL;
	(* Variables allocation *)
	VAR_Pointer : POINTER TO ARRAY[0..99] OF WORD;
	VAR_Cfg		: POINTER TO typ_MODBUS_VAR;
END_VAR
VAR_OUTPUT
	(* Status *)
	Status_Log	: BYTE;
	Status_Vis	: DWORD;
END_VAR
VAR
	sta         : BYTE :=0;
	i			: BYTE;
	j			: BYTE;
	Alarm		: FLT_EVENT;

	VarTmr		: TON := (PT:=T#1s);
	VarSta		: BYTE; (* Status *)
	VarCnt		: BYTE; (* Scan counter *)
	VarRetry	: BYTE;
	VarAlarm	: BYTE; (* Last variable with errors *)
END_VAR
MB_MASTER( strIP_ADDRESS:=IP, wPORT:=PORT, tTIME_OUT:=T#750MS, (*xCONNECT:=TRUE,*)
		   ptREAD_DATA:=ADR(MB_READBUF), ptSEND_DATA:=ADR(MB_WRITEBUF), xSEND:=MB_Start );

IF sta=0 THEN
	MB_MASTER.xCONNECT:=TRUE;
	sta:=1;
END_IF

(* Process variable management *)
IF VARS_En THEN VARS_Process(); END_IF





(* Check status *)
Alarm(IN:=(MB_MASTER.wERROR<>0));
IF Alarm.EVH THEN
	LogEv(SEL(MB_MASTER.wERROR>0,EL_Wrn,EL_Alarm),EO_MODBUS_TCP,ID,1,WORD_TO_STRING(MB_MASTER.wERROR));
END_IF
IF Alarm.EVL THEN
	LogEv(EL_Log,EO_MODBUS_TCP,ID,2,'');
END_IF

(* Log/visu status *)
   IF Alarm.IN   THEN Status_Log:=2; Status_Vis:=COLOR_RED;
ELSIF Vars_Alarm THEN Status_Log:=1; Status_Vis:=COLOR_YELLOW;
  				 ELSE Status_Log:=0; Status_Vis:=COLOR_GREEN;
END_IF
END_FUNCTION_BLOCK
ACTION VAR_Search:
(* Search VAR with specific pointer if not found return first free VAR
	[Last VAR is not active... used as safe area...] 
*)
j:=VARS_Max;
FOR i := 0 TO VARS_Max-1 DO
	IF VARS[i].Variable=0 AND j>i THEN j:=i; END_IF
	IF VARS[i].Variable=VAR_Pointer THEN
		VAR_Cfg:=ADR(VARS[i]);
		RETURN;
	END_IF
END_FOR
VAR_Cfg:=ADR(VARS[j]);
END_ACTION
ACTION VARS_Process:
(* Update var timers *)
VarTmr(IN:=(NOT VarTmr.Q));
IF VarTmr.Q THEN
	FOR i := 0 TO VARS_Max DO
		IF VARS[i].Refresh_Cnt>0 THEN VARS[i].Refresh_Cnt:=VARS[i].Refresh_Cnt-1; END_IF
	END_FOR
	VARS_Check:=TRUE;
END_IF


(* Process status *)
CASE VarSta OF
	0: (* === Init *)
		VarCnt:=0;
		VarSta:=1;

	1: (* === Wait check signal *)
		IF VARS_Check THEN
			VARS_Check:=FALSE;
			VarCnt:=0;
			VarSta:=2;
		END_IF

	2: (* === Check loop *)
		IF NOT (MB_Lock OR MB_Start) THEN
			WHILE VarCnt<=(VARS_Max-1) AND VarSta=2 DO
				(* Check only active vars *)
				IF VARS[VarCnt].Variable<>0 THEN
					(* Check var auto-refresh on timer checks *)
					IF VARS[VarCnt].Refresh_Time>0 AND VARS[VarCnt].Refresh_Cnt=0 THEN
						VARS[VarCnt].Refresh_Cnt:=VARS[VarCnt].Refresh_Time;
						VarSta:=3;
					END_IF
					(* Check refresh for change or request *)
					CASE VARS[VarCnt].FunCode OF
						5,6,15,16: (* Write functions *)
							IF VARS[VarCnt].Variable_Size=1 THEN
								IF VARS[VarCnt].Variable^<>VARS[VarCnt].Variable_Mirror THEN
									VARS[VarCnt].Variable_Mirror:=VARS[VarCnt].Variable^;
									VarSta:=3;
								END_IF
							ELSE
								IF VARS[VarCnt].Variable_Mirror<>0 THEN
									VARS[VarCnt].Variable_Mirror:=0;
									VarSta:=3;
								END_IF
							END_IF
						1,2,3,4: (* Write functions *)
							IF VARS[VarCnt].Variable_Mirror<>0 THEN
								VARS[VarCnt].Variable_Mirror:=0;
								VarSta:=3;
							END_IF
					END_CASE
				END_IF
				(* Process query *)
				IF VarSta=3 THEN
					MB_Lock:=TRUE;
					MB_MASTER.bUNIT_ID:=VARS[VarCnt].SlaveAddress;
					MB_MASTER.bFUNCTION_CODE:=VARS[VarCnt].FunCode;
					CASE VARS[VarCnt].FunCode OF
						16#5,16#6,16#F,16#10:
							MB_MASTER.wREAD_ADDRESS:=0;
							MB_MASTER.wREAD_QUANTITY:=0;
							MB_MASTER.wWRITE_ADDRESS:=VARS[VarCnt].FunAddress;
							MB_MASTER.wWRITE_QUANTITY:=VARS[VarCnt].Variable_Size;
							IF VARS[VarCnt].Variable_Size=200 THEN
								COPY_32SWAP16(VARS[VarCnt].Variable, ADR(MB_WRITEBUF));
							ELSIF VARS[VarCnt].Variable_Size>1 THEN
								MEMCPY(VARS[VarCnt].Variable, ADR(MB_WRITEBUF), 2*VARS[VarCnt].Variable_Size);
							ELSE
								MB_WRITEBUF[0]:=VARS[VarCnt].Variable^;
							END_IF
						16#1,16#2,16#3,16#4:
							MB_MASTER.wREAD_ADDRESS:=VARS[VarCnt].FunAddress;
							IF VARS[VarCnt].Variable_Size=200 THEN MB_MASTER.wREAD_QUANTITY:=2; ELSE
							  MB_MASTER.wREAD_QUANTITY:=VARS[VarCnt].Variable_Size;
							END_IF
							MB_MASTER.wWRITE_ADDRESS:=0;
							MB_MASTER.wWRITE_QUANTITY:=0;
					END_CASE
					VarRetry:=0;
					MB_Start:=TRUE;
				ELSE
					VarCnt:=VarCnt+1;
				END_IF
			END_WHILE
			(* Check loop completed -> no actions *)
			IF VarSta=2 THEN VarSta:=1; END_IF
		END_IF

	3: (* === Wait & process MB response *)
		IF NOT MB_Start THEN
			IF MB_MASTER.wERROR=0 THEN
				CASE VARS[VarCnt].FunCode OF
					1,2,3,4:
						IF VARS[VarCnt].Variable_Size=200 THEN
							COPY_32SWAP16(ADR(MB_READBUF), VARS[VarCnt].Variable);
						ELSIF VARS[VarCnt].Variable_Size>1 THEN
							MEMCPY(ADR(MB_READBUF), VARS[VarCnt].Variable, 2*VARS[VarCnt].Variable_Size);
						ELSE
							VARS[VarCnt].Variable^:=MB_READBUF[0];
						END_IF
				END_CASE
				MB_Lock:=FALSE;
				(* Signal error recovery *)
				IF VARS_Alarm=TRUE AND VarCnt=VarAlarm THEN
					LogEv(EL_Wrn,EO_MODBUS_TCP,ID,5,'');
					VARS_Alarm:=FALSE;
				END_IF
				(* Next var *)
				VarCnt:=VarCnt+1;
				VarSta:=2;
			ELSE
				IF VarRetry<10 THEN
					VarRetry:=VarRetry+1;
					MB_Start:=TRUE;
				ELSE
					MB_Lock:=FALSE;
					(* Signal error *)
					IF VARS_Alarm=FALSE THEN
						LogEv(EL_Wrn,EO_MODBUS_TCP,ID,3,WORD_TO_STRING(MB_MASTER.wERROR));
						VARS_Alarm:=TRUE;
						VarAlarm:=VarCnt-1;
					END_IF
					(* Next var *)
					VarCnt:=VarCnt+1;
					VarSta:=2;
				END_IF
			END_IF
		END_IF

ELSE
	VarSta:=0;
END_CASE
END_ACTION

(* POU Plant_Objects/obj_TPV, ST *)
FUNCTION_BLOCK obj_TPV
(* === TEMPERATURE PROBE  ===
   v1.0[16/04/15] - Versioning
*)
VAR CONSTANT
	NormalEv		: BYTE := 0;
	ErrorEv			: BYTE := 1;
	WarningEv		: BYTE := 2;
END_VAR
VAR_INPUT
	(* Settings *)
	ID				: BYTE;
	TAP				: BYTE:=4;	   (* Consecutive checks filter *)
	INITEV			: BOOL:= TRUE; (* Generate init OK event *)
	IN_EMIN			: INT :=-2000; (* Low error limit *)
	IN_WMIN			: INT := -550; (* Low warning value *)
	IN_WMAX			: INT :=  900; (* High warning value *)
	IN_EMAX			: INT := 8500; (* High error limit *)
	ERR_MIN_SHORT	: BOOL:= TRUE; (* TRUE  ==> EMIN=Short        , EMAX=Disconnected
									  FALSE ==> EMIN=Disconnected , EMAX=Short 		 *)
	(* Physical input *)
	IN			: INT;
END_VAR
VAR_OUTPUT
	WRN			: BOOL;	(* Value in warning range *)
	ERR			: BOOL;	(* Value error *)
	HI			: INT;	(* Highest value - cleared by Stat_Reset() action *)
	AVG			: INT; 	(* Average value - updated by Mean() action, cleared by Mean_Reset() action *)
	LOW			: INT;	(* Lowest value  - cleared by Stat_Reset() action *)

	Status_Log	: WORD;
	Status_Vis	: DWORD;
END_VAR
VAR
	cnt			: BYTE;
	event		: BYTE := 0;	(* 0: monitoring a generic, 1: monitoring an error, 2: monitoring a warning *)
	asum		: DINT;
	acnt		: WORD;
END_VAR
(* Check probe value limits *)
IF IN<=IN_EMIN OR IN>=IN_EMAX THEN
	IF NOT ERR THEN
		IF event <> ErrorEv THEN
			cnt := 1;
			event := ErrorEv;
		ELSE
			cnt:=cnt+1;
		END_IF

		IF cnt>TAP THEN
			cnt:=0;
			ERR:=TRUE; WRN:=FALSE;
			IF ( ERR_MIN_SHORT=TRUE  AND IN<=IN_EMIN ) OR ( ERR_MIN_SHORT=FALSE AND IN>=IN_EMAX ) THEN
				LogEv(EL_Alarm,EO_TPV,ID,5,INT_TO_STRING(IN));
			ELSE
				LogEv(EL_Alarm,EO_TPV,ID,4,INT_TO_STRING(IN));
			END_IF
		END_IF
	END_IF
ELSIF IN<=IN_WMIN OR IN>=IN_WMAX THEN
	IF NOT WRN THEN
		IF event <> WarningEv THEN
			cnt := 1;
			event := WarningEv;
		ELSE
			cnt:=cnt+1;
		END_IF

		IF cnt>TAP THEN
			cnt:=0;
			ERR:=FALSE; WRN:=TRUE;
			LogEv(EL_Wrn,EO_TPV,ID,SEL(IN<=IN_WMIN,3,2),INT_TO_STRING(IN));
		END_IF
	END_IF
ELSE
	IF INITEV OR WRN OR ERR THEN
		IF event <> NormalEv THEN
			cnt := 1;
			event := NormalEv;
		ELSE
			cnt:=cnt+1;
		END_IF

		IF cnt>TAP THEN
			cnt:=0;
			INITEV:=FALSE; ERR:=FALSE; WRN:=FALSE;
			LogEv(EL_Log,EO_TPV,ID,1,'Probe_OK');
		END_IF
	END_IF
END_IF

(* Average value *)
IF acnt>=500 THEN
	Mean();
	asum := asum - AVG;
	acnt := acnt - 1;
END_IF

asum := asum + IN;
acnt := acnt + 1;

(* Statistics values *)
IF IN<LOW THEN LOW:=IN; END_IF
IF IN>HI  THEN HI :=IN; END_IF

Lamp.obj_Status := Status_Log;
Lamp.UpdateStatus();

(* Status Log *)
IF ERR THEN	Status_Log := 2; Status_Vis := COLOR_RED;
ELSIF WRN THEN Status_Log := 1;	Status_Vis := COLOR_YELLOW;
ELSE Status_Log := 0; Status_Vis := COLOR_GREEN;
END_IF
END_FUNCTION_BLOCK
ACTION AddLogData:
Logger.s1:=INSERT('&TPV=',BYTE_TO_STRING(ID),4);
IF ID<10 THEN Logger.s1:=INSERT(Logger.s1,'0',4); END_IF

Mean();

Logger.s1:=CONCAT(Logger.s1,INT_TO_STRING(AVG));		Logger.s1:=CONCAT(Logger.s1,';');

Logger.s1:=CONCAT(Logger.s1,WORD_TO_STRING(Status_Log));
ADDSTRING(ADR(Logger.TData), ADR(Logger.s1), Logger.TLen);
END_ACTION
ACTION Mean:
AVG := DINT_TO_INT(asum/acnt);
END_ACTION
ACTION Mean_Reset:
AVG:=IN;
asum:=IN;
acnt:=1;
END_ACTION
ACTION Stat_Reset:
HI:=IN;
LOW:=IN;
END_ACTION

(* POU Plant_Objects/obj_VRD_new, ST *)
FUNCTION_BLOCK obj_VRD_new
(* === VALVOLA RIPARTITORE ===
   v1.0[16/04/15] - Versioning
*)
VAR CONSTANT
	Chk_CntSecAlarm	: INT := 900;	(* 900s = 15 minutes -> Observation itme *)
END_VAR
VAR_INPUT
	(* Settings *)
	ID				: BYTE;
	(* Controls *)
	RUN  			: BOOL;					(* Control input *)
	ReducedRange	: BOOL := FALSE;		(* If true output value is among 2 and 10V, otherwise 0-10V *)

	(* Physical inputs *)
	TEMP 			: INT;		(* Input temperature from sensor *)
	STATUS 			: WORD;		(* Input position from valve *)

	InitOK			: BOOL;
	Alarm1			: BOOL;
	Alarm2			: BOOL;
	Warning			: BOOL;

	Ctrl_Init		: BOOL;
	Ctrl_SetPoint	: INT;
	Ctrl_SetPointNew: INT := 0;
	Delta_SetPoint	: INT;
	Ctrl_Err		: INT;			(* Current error *)
	Ctrl_Err0		: INT; 			(* Previous error *)
	Ctrl_Accel		: REAL;			(* Derivate of error *)
	Ctrl_AccelGate  : INT:=1;		(* Derivate gate *)
	Ctrl_AccelTmr	: WORD;
	Ctrl_SetPointGate: INT := 5;	(* Setpoint gate - 0.5°C *)
	Ctrl_ErrGate	: INT:=5;		(* Error gate *)
	Ctrl_Kp			: REAL:=2;(*1;*)		(* Proportional factor *)
	Ctrl_Kd			: REAL:=10;(*100;*)  	(* Derivative factor *)
	Ctrl_Out		: REAL;

	Chk_Err			: INT;
	Chk_ErrGate		: INT:=1000; 			(* Check error gate *)
	Chk_Cnt			: INT;
	Chk_CntAlarm	: INT:=240; 		(* Check error trigger 120s *)

	(* Status *)
	Log_AvgTemp		: AVERAGE_T;
	Status_Log		: BYTE;
	Status_Vis 		: DWORD;

	(* Feedback *)
	fFeedback		: BOOL;			(* TRUE: Feedback available, FALSE: Feedback not available *)

END_VAR
VAR_IN_OUT
	CLIM		: typ_Clima;
END_VAR
VAR_OUTPUT
	(* Physical outputs *)
	OUT			: WORD;
END_VAR
VAR
	Curve		: CHARCURVE;
	Curve_Err	: BYTE;

	aTemp		: ARRAY [1..20] OF INT;
	meanTemp	: INT;
	sum			: INT := 0;
	Tmr			: TON := (PT:=T#1s);
	index		: BYTE;
	i			: BYTE;
	fCtrl_Err	: BOOL;		(* TRUE: Ctrl_Err>0, FALSE: Ctrl_Err<0 *)

END_VAR

VAR_INPUT RETAIN
	Local_VRD_TAlarm: INT;
END_VAR
(* Check initialization *)
(*IF NOT InitOK THEN Init(); END_IF*)

(* Check max temperature *)
IF TEMP>Local_VRD_TAlarm THEN
	IF NOT Alarm1 THEN
		Alarm1:=TRUE;
		LogEv(EL_AlarmStop,EO_VRD,ID,3,'VRD_Overtemperature');
	END_IF
END_IF

IF (TEMP<Local_VRD_TAlarm-100) AND Alarm1  THEN
		Alarm1:=FALSE;
END_IF

(* Check climatic setup *)
IF NOT CLIM.InitOK THEN	DefaultClim(); END_IF;
(* Calculate Setpoint *)
Curve(	IN:= T_AMB,	N:= 5, P:= CLIM.Points,			(* Given the x value as input, the corresponding y value as output is returned, if it matches the crve designed by array of points *)
		OUT=> Ctrl_SetPointNew, ERR=> Curve_Err );

IF Curve_Err>0 OR Ctrl_SetPoint>Plant_VRD_TMax THEN
	Ctrl_SetPoint:=Plant_VRD_TDefault;
	IF NOT Warning THEN
		Warning:=TRUE;
		LogEv(EL_Wrn,EO_VRD,ID,2,'VRD_Climatic_Error');
	END_IF
ELSE
	Delta_SetPoint := ABS(Ctrl_SetPoint - Ctrl_SetPointNew);
	IF Delta_SetPoint>Ctrl_SetPointGate THEN Ctrl_SetPoint := Ctrl_SetPointNew; END_IF

	Warning:=FALSE;
END_IF

(* Execute control loop [T=500ms] *)
IF RUN AND (NOT Alarm1) THEN
	(* Calculate error *)
	Ctrl_Err:=Ctrl_SetPoint-TEMP;
	(* Init/restart operations *)
	IF NOT Ctrl_Init THEN
		Ctrl_Accel:=0;
		Ctrl_AccelTmr:=0;
		Ctrl_Err0:=Ctrl_Err;
		Ctrl_Out:=5000;
		Ctrl_Init:=TRUE;
	END_IF
	(* Calculate acceleration *)
	IF ABS(Ctrl_Err-Ctrl_Err0)>Ctrl_AccelGate OR Ctrl_AccelTmr>20 THEN
		Ctrl_Accel:=INT_TO_REAL(Ctrl_Err-Ctrl_Err0)/WORD_TO_REAL(1+Ctrl_AccelTmr);
		Ctrl_AccelTmr:=0;
		Ctrl_Err0:=Ctrl_Err;
	ELSE
		Ctrl_AccelTmr:=Ctrl_AccelTmr+1;
	END_IF

	(* Gate error *)
	IF ABS(Ctrl_Err)>Ctrl_ErrGate THEN
		(* Control loop *)
		Ctrl_Out:=Ctrl_Out+(Ctrl_Kp*Ctrl_Err)+(Ctrl_Kd*Ctrl_Accel);
	END_IF

	(* Limiter and Output *)
(*	Ctrl_Out:=LIMIT(0,Ctrl_Out,27000); *)
	Ctrl_Out:=LIMIT(0,Ctrl_Out,32766);

	OUT:=REAL_TO_WORD(Ctrl_Out);

ELSE
	Ctrl_Init:=FALSE;
	OUT:=0;
END_IF

(* If there is an hardware feedback (such as 0-10V, potentiometer, ...) check it otherwise try to rebuild it *)
IF fFeedback THEN CheckFeedback();
ELSE BuildFeedback();
END_IF

(* Status temp *)
Log_AvgTemp(IN:=Temp);
Lamp.UpdateStatus(obj_Status := Status_Log);

(* Status color *)
   IF Alarm1  THEN Status_Log:=2; Status_Vis:=16#2020F0;
ELSIF Warning OR Alarm2        THEN Status_Log:=1; Status_Vis:=16#20F0F0;
                       ELSE Status_Log:=0; Status_Vis:=SEL(RUN,16#006000,16#20F020);
END_IF
END_FUNCTION_BLOCK
ACTION AddLogData:
Logger.s1:=INSERT('&VRD=',BYTE_TO_STRING(ID),4);
IF ID<10 THEN Logger.s1:=INSERT(Logger.s1,'0',4); END_IF

Logger.s1:=CONCAT(Logger.s1,INT_TO_STRING(Ctrl_SetPoint));				Logger.s1:=CONCAT(Logger.s1,';');
Logger.s1:=CONCAT(Logger.s1,WORD_TO_STRING(OUT/327));						Logger.s1:=CONCAT(Logger.s1,';');

IF fFeedback THEN Logger.s1:=CONCAT(Logger.s1,WORD_TO_STRING(STATUS));
ELSE Logger.s1:=CONCAT(Logger.s1,'0');	(* Bypass *)
END_IF

Logger.s1:=CONCAT(Logger.s1,';');

Logger.s1:=CONCAT(Logger.s1,WORD_TO_STRING(Status_Log));

Logger.s1:=CONCAT(Logger.s1,';');
Logger.s1:=CONCAT(Logger.s1,'1'); (* Valvola modulante controllata Analogica *)

ADDSTRING(ADR(Logger.TData), ADR(Logger.s1), Logger.TLen);
END_ACTION
ACTION BuildFeedback:
(* Comparison is taken between actual temperature vs windowed mean value of last 20 temperature
   (check is carried out every second)	*)
IF RUN AND (NOT Alarm1) THEN

	IF Ctrl_Err>0 THEN
		IF NOT fCtrl_Err THEN index := 0; END_IF
		fCtrl_Err := TRUE;
	ELSE
		IF fCtrl_Err THEN index := 0; END_IF
		fCtrl_Err := FALSE;
	END_IF

	(* Temperature is lower than setpoint -->> Should increase *)
	Tmr(IN:=NOT Tmr.Q);

	IF Tmr.Q THEN

		IF index<21 THEN
			(* Fullfil temperature array *)
			aTemp[index] := TEMP;
			index := index + 1;

			IF index=20 THEN
				FOR i:=1 TO 20 BY 1 DO sum := sum + aTemp[i]; END_FOR
			END_IF
		ELSE
			(* Calculate mean value *)
			meanTemp := sum/20;

			IF (fCtrl_Err AND TEMP<meanTemp) OR (NOT fCtrl_Err AND TEMP>meanTemp) THEN

				IF Chk_Cnt>Chk_CntSecAlarm THEN
					IF NOT Alarm2 THEN
						Alarm2:=TRUE;
						LogEv(EL_Alarm,EO_VRD,ID,4,'VRD_Position_Error');
					END_IF
				ELSE
					Chk_Cnt := Chk_Cnt+1;
				END_IF

			ELSE
				(* Reset counter and alarm flag *)
				Chk_Cnt:=0;
				Alarm2:=FALSE;
			END_IF

			sum := 0;	(* Reset sum counter *)

			(* Shift array removing oldest value *)
			FOR i:=1 TO 20 BY 1 DO
				aTemp[i-1] := aTemp[i];
				sum := sum + aTemp[i];
			END_FOR

			aTemp[20] := TEMP;			(* Last temperature value is new one *)
			sum := sum + aTemp[20];		(* Update sum *)
		END_IF
	END_IF
END_IF
END_ACTION
ACTION CheckFeedback:
(* Calculate position error according to feedback *)
IF ReducedRange THEN
(* SETPOINT[2..10V]-STATUS[0..10V] *)
	IF OUT<=6553 THEN Chk_Err:=0; ELSE Chk_Err:=(OUT-6553)/262; END_IF
	Chk_Err:=(Chk_Err-STATUS)/327;
ELSE
(* SETPOINT[0..10V]-STATUS[0..10V] *)
	Chk_Err := OUT - STATUS;
END_IF

(* Check position error *)
IF ( ABS(Chk_Err)>Chk_ErrGate ) THEN
	IF Chk_Cnt>Chk_CntAlarm THEN
		IF NOT Alarm2 THEN
			Alarm2:=TRUE;
			LogEv(EL_Wrn,EO_VRD,ID,4,'VRD_Position_Error');
		END_IF
	ELSE
		Chk_Cnt:=Chk_Cnt+1;
	END_IF
ELSE
	Chk_Cnt:=0;
	Alarm2:=FALSE;
END_IF
END_ACTION
ACTION DefaultClim:
(*CLIM.Points[0].X:=-300; CLIM.Points[0].Y:=400;
CLIM.Points[1].X:=-50;  CLIM.Points[1].Y:=400;
CLIM.Points[2].X:= 200; CLIM.Points[2].Y:=200;
CLIM.Points[3].X:= 300; CLIM.Points[3].Y:=200;
CLIM.Points[4].X:= 500; CLIM.Points[4].Y:=200;*)
CLIM.Points[0].X:=-300; CLIM.Points[0].Y:=850;
CLIM.Points[1].X:=-50;  CLIM.Points[1].Y:=650;
CLIM.Points[2].X:= 100; CLIM.Points[2].Y:=400;
CLIM.Points[3].X:= 200; CLIM.Points[3].Y:=200;
CLIM.Points[4].X:= 500; CLIM.Points[4].Y:=200;
CLIM.InitOK:=TRUE;
LogEv(EL_Wrn,EO_VRD,ID,1,'Climatic_Default');
END_ACTION
ACTION Init:
(* End initialization *)
InitOK:=TRUE;
END_ACTION

(* POU Plant_Objects/obj_VRD_POT_new, ST *)
FUNCTION_BLOCK obj_VRD_POT_new
(* === VALVOLA RIPARTITORE ===
   v1.0[16/04/15] - Versioning
*)
VAR CONSTANT
	ValveOpenRes	: WORD := 16#07D0;
	ValveCloseRes	: WORD := 16#EC00;

	ValvePosCheck	: BYTE :=4;

	Chk_CntSecAlarm	: INT := 900;	(* 900s = 15 minutes -> Observation itme *)
END_VAR
VAR_INPUT
	(* Settings *)
	ID				: BYTE;
	(* Controls *)
	RUN  			: BOOL;		(* Control input *)

	(* Physical inputs *)
	TEMP 			: INT;		(* Input temperature from sensor *)
	STATUS 			: WORD;		(* Input position from valve *)

	InitOK			: BOOL;
	Alarm1			: BOOL;
	Alarm2			: BOOL;
	Warning			: BOOL;

	Ctrl_Init		: BOOL;
	Ctrl_SetPoint	: INT;
	Ctrl_SetPointNew: INT := 0;
	Delta_SetPoint	: INT;
	Ctrl_Err		: INT;			(* Current error *)
	Ctrl_Err0		: INT; 			(* Previous error *)
	Ctrl_Accel		: REAL;			(* Derivate of error *)
	Ctrl_AccelGate  : INT:=1;		(* Derivate gate - 0.1°C/500ms *)
	Ctrl_AccelTmr	: WORD;
	Ctrl_SetPointGate: INT := 5;	(* Setpoint gate - 0.5°C *)
	Ctrl_ErrGate	: INT:=5;		(* Error gate - 0.5°C *)
	Ctrl_Kp			: REAL:=1;(*5;*)		(* Proportional factor *)
	Ctrl_Kd			: REAL:=5;(*10;*)  	(* Derivative factor *)
	Ctrl_Out		: REAL;

	(*Chk_Err			: INT;	*)
	Chk_Err			: REAL;
	Chk_ErrGate		: INT:=1000; 		(* Check error gate *)
	Chk_Cnt			: INT;
	Chk_CntAlarm	: INT:=60; 			(* Check error trigger 60s *)

	(* Status *)
	Log_AvgTemp		: AVERAGE_T;

	(* Control parameters *)
	Tpwm			: TIME := T#2s;

	(* Feedback *)
	fFeedback		: BOOL;			(* TRUE: Feedback available, FALSE: Feedback not available *)

END_VAR
VAR_IN_OUT
	CLIM		: typ_Clima;
END_VAR
VAR_OUTPUT
	(* Physical outputs *)
	OUT_CL		: BOOL;
	OUT_OP		: BOOL;

	Status_Log		: BYTE;
	Status_Vis 		: DWORD;
END_VAR
VAR
	Curve		: CHARCURVE;
	Curve_Err	: BYTE;

	Ctrl_Out_Time	:	REAL;
	PwmTmr			:   TON := (PT:=T#5s);

	fClose		: BOOL;	(* Valve is completly closed *)
	fOpen		: BOOL;	(* Valve is completely open  *)
	CloseCtr	: BYTE;	(* Close counter *)
	OpenCtr		: BYTE; (* Open counter  *)

	aTemp		: ARRAY [1..20] OF INT;
	meanTemp	: INT;
	sum			: INT := 0;
	Tmr			: TON := (PT:=T#1s);
	index		: BYTE;
	i			: BYTE;
	fCtrl_Err	: BOOL;		(* TRUE: Ctrl_Err>0, FALSE: Ctrl_Err<0 *)
END_VAR

VAR_INPUT RETAIN
	Local_VRD_TAlarm: INT;
END_VAR
(* Check initialization *)
IF NOT InitOK THEN Init(); END_IF

(* Check max temperature *)
IF TEMP>Local_VRD_TAlarm THEN
	IF NOT Alarm1 THEN
		Alarm1:=TRUE;
		LogEv(EL_AlarmStop,EO_VRD,ID,3,'VRD_Overtemperature');
	END_IF
END_IF

IF (TEMP<Local_VRD_TAlarm-100) AND Alarm1  THEN
		Alarm1:=FALSE;
END_IF

(* Check climatic setup *)
IF NOT CLIM.InitOK THEN	DefaultClim(); END_IF;
(* Calculate Setpoint *)
Curve(	IN:= T_AMB,	N:= 5, P:= CLIM.Points,			(* Given the x value as input, the corresponding y value as output is returned, if it matches the crve designed by array of points *)
		OUT=> Ctrl_SetPointNew, ERR=> Curve_Err );
IF Curve_Err>0 OR Ctrl_SetPoint>Plant_VRD_TMax THEN
	Ctrl_SetPoint:=Plant_VRD_TDefault;
	IF NOT Warning THEN
		Warning:=TRUE;
		LogEv(EL_Wrn,EO_VRD,ID,2,'VRD_Climatic_Error');
	END_IF
ELSE
	Delta_SetPoint := ABS(Ctrl_SetPoint - Ctrl_SetPointNew);
	IF Delta_SetPoint>Ctrl_SetPointGate THEN Ctrl_SetPoint := Ctrl_SetPointNew; END_IF

	Warning:=FALSE;
END_IF

(* Execute control loop [T=500ms] *)
IF RUN AND (NOT Alarm1) THEN
	(* Calculate error *)
	Ctrl_Err:=Ctrl_SetPoint-TEMP;
	(* Init/restart operations *)
	IF NOT Ctrl_Init THEN
		Ctrl_Accel:=0;
		Ctrl_AccelTmr:=0;
		Ctrl_Err0:=Ctrl_Err;
		Ctrl_Out:=0;
		Ctrl_Init:=TRUE;
	END_IF
	(* Calculate acceleration *)
	IF ABS(Ctrl_Err-Ctrl_Err0)>Ctrl_AccelGate OR Ctrl_AccelTmr>2 THEN
		Ctrl_Accel:=INT_TO_REAL(Ctrl_Err-Ctrl_Err0)/WORD_TO_REAL(1+Ctrl_AccelTmr);
		Ctrl_AccelTmr:=0;
		Ctrl_Err0:=Ctrl_Err;
	ELSE
		Ctrl_AccelTmr:=Ctrl_AccelTmr+1;
	END_IF

	(* Gate error *)
	IF ABS(Ctrl_Err)>Ctrl_ErrGate THEN
		(* Control loop *)
		Ctrl_Out:=Ctrl_Out+(Ctrl_Kp*Ctrl_Err)+(Ctrl_Kd*Ctrl_Accel);

		(* Limiter and Output *)
		Ctrl_Out_Time := LIMIT(0,ABS(Ctrl_Out),TIME_TO_REAL(Tpwm));

		PwmTmr(IN:=NOT PwmTmr.Q);

		IF PwmTmr.ET>=REAL_TO_TIME(Ctrl_Out_Time) THEN
			(* Stop corretction *)
			OUT_OP := FALSE;
			OUT_CL := FALSE;
		END_IF

		IF PwmTmr.Q THEN
			(* Adjust valve position *)
			IF fFeedback THEN
				IF Ctrl_Err>0 AND NOT fOpen THEN OUT_OP := TRUE; END_IF		(* If valve yet open don't drive physical output *)
				IF Ctrl_Err<0 AND NOT fClose THEN OUT_CL := TRUE; END_IF	(* If valve yet close don't drive physical output *)
			ELSE
				IF Ctrl_Err>0 THEN OUT_OP := TRUE; END_IF
				IF Ctrl_Err<0 THEN OUT_CL := TRUE; END_IF
			END_IF

			PwmTmr.PT := Tpwm;
		END_IF
	END_IF
ELSE
	OUT_CL := TRUE;
	OUT_OP := FALSE;		(* forzatura serranda in chiusura se il circolatore corrispettivo non è comandato *)
	Ctrl_Init:=FALSE;
END_IF

(* If there is an hardware feedback (such as 0-10V, potentiometer, ...) check it otherwise try to rebuild it *)
IF fFeedback THEN CheckFeedback();
ELSE BuildFeedback();
END_IF

(* Status temp *)
Log_AvgTemp(IN:=Temp);
Lamp.UpdateStatus(obj_Status := Status_Log);

(* Status color *)
   IF Alarm1 THEN Status_Log:=2; Status_Vis:=COLOR_RED;
ELSIF Warning  OR Alarm2         THEN Status_Log:=1; Status_Vis:=COLOR_YELLOW;
                       ELSE Status_Log:=0; Status_Vis:=SEL(RUN,COLOR_LIGHT_GREEN,COLOR_GREEN);
END_IF
END_FUNCTION_BLOCK
ACTION AddLogData:
Logger.s1:=INSERT('&VRD=',BYTE_TO_STRING(ID),4);
IF ID<10 THEN Logger.s1:=INSERT(Logger.s1,'0',4); END_IF

Logger.s1:=CONCAT(Logger.s1,INT_TO_STRING(Ctrl_SetPoint));
Logger.s1:=CONCAT(Logger.s1,';');
Logger.s1:=CONCAT(Logger.s1,'0');	(* Bypass *)
Logger.s1:=CONCAT(Logger.s1,';');

IF fFeedback THEN Logger.s1:=CONCAT(Logger.s1,WORD_TO_STRING(STATUS));
ELSE Logger.s1:=CONCAT(Logger.s1,'0');	(* Bypass *)
END_IF

Logger.s1:=CONCAT(Logger.s1,WORD_TO_STRING(Status_Log));

Logger.s1:=CONCAT(Logger.s1,';');
Logger.s1:=CONCAT(Logger.s1,'0'); (* Valvola modulante controllata digitale *)

Logger.s1:=CONCAT(Logger.s1,';');
Logger.s1:=CONCAT(Logger.s1,SEL(OUT_OP,'0','100'));
Logger.s1:=CONCAT(Logger.s1,';');
Logger.s1:=CONCAT(Logger.s1,SEL(OUT_CL,'0','100'));




ADDSTRING(ADR(Logger.TData), ADR(Logger.s1), Logger.TLen);
END_ACTION
ACTION BuildFeedback:
(* Comparison is taken between actual temperature vs windowed mean value OF last 20 temperature
   (check is carried out every second)	*)
IF RUN AND (NOT Alarm1) THEN

	IF Ctrl_Err>0 THEN
		IF NOT fCtrl_Err THEN index := 0; END_IF
		fCtrl_Err := TRUE;
	ELSE
		IF fCtrl_Err THEN index := 0; END_IF
		fCtrl_Err := FALSE;
	END_IF

	(* Temperature is lower than setpoint -->> Should increase *)
	Tmr(IN:=NOT Tmr.Q);

	IF Tmr.Q THEN

		IF index<21 THEN
			(* Fullfil temperature array *)
			aTemp[index] := TEMP;
			index := index + 1;

			IF index=20 THEN
				FOR i:=1 TO 20 BY 1 DO sum := sum + aTemp[i]; END_FOR
			END_IF
		ELSE
			(* Calculate mean value *)
			meanTemp := sum/20;

			IF (fCtrl_Err AND TEMP<meanTemp) OR (NOT fCtrl_Err AND TEMP>meanTemp) THEN

				IF Chk_Cnt>Chk_CntSecAlarm THEN
					IF NOT Alarm2 THEN
						Alarm2:=TRUE;
						LogEv(EL_Alarm,EO_VRD,ID,4,'VRD_Position_Error');
					END_IF
				ELSE
					Chk_Cnt := Chk_Cnt+1;
				END_IF

			ELSE
				(* Reset counter and alarm flag *)
				Chk_Cnt:=0;
				Alarm2:=FALSE;
			END_IF

			sum := 0;	(* Reset sum counter *)

			(* Shift array removing oldest value *)
			FOR i:=1 TO 20 BY 1 DO
				aTemp[i-1] := aTemp[i];
				sum := sum + aTemp[i];
			END_FOR

			aTemp[20] := TEMP;			(* Last temperature value is new one *)
			sum := sum + aTemp[20];		(* Update sum *)
		END_IF
	END_IF
END_IF
END_ACTION
ACTION CheckFeedback:
(* Check position *)
IF Status=ValveCloseRes THEN

	CloseCtr := CloseCtr+1;
	IF CloseCtr=ValvePosCheck THEN	fClose := TRUE;	END_IF

ELSIF Status=ValveOpenRes THEN

	OpenCtr := OpenCtr+1;
	IF OpenCtr=ValvePosCheck THEN	fOpen := TRUE;	END_IF

ELSE

	fClose := FALSE;
	fOpen  := FALSE;

END_IF

(* Check position error *)


(* 0xEC00 corresponds to 0ohm, while other values are linear from 20 (10ohm -> 1%) to 2000 (1Kohm -> 100%) *)
IF Status = 16#EC00 THEN Chk_Err := Ctrl_Out;
ELSE
   Chk_Err := Ctrl_Out - Status/2;
END_IF

IF ( Chk_Err<-Chk_ErrGate OR Chk_Err>Chk_ErrGate ) THEN
	IF Chk_Cnt>Chk_CntAlarm THEN
		IF NOT Alarm2 THEN
			Alarm2:=TRUE;
			LogEv(EL_Wrn,EO_VRD,ID,4,'VRD_Position_Error');
		END_IF
	ELSE
		Chk_Cnt:=Chk_Cnt+1;
	END_IF
ELSE
	Chk_Cnt:=0;
	Alarm2:=FALSE;
END_IF
END_ACTION
ACTION DefaultClim:
CLIM.Points[0].X:=-300; CLIM.Points[0].Y:=850;
CLIM.Points[1].X:=-70;  CLIM.Points[1].Y:=750;
CLIM.Points[2].X:= 100; CLIM.Points[2].Y:=630;
CLIM.Points[3].X:= 200; CLIM.Points[3].Y:=250;
CLIM.Points[4].X:= 500; CLIM.Points[4].Y:=200;
CLIM.InitOK:=TRUE;
LogEv(EL_Wrn,EO_VRD,ID,1,'Climatic_Default');
END_ACTION
ACTION Init:
(* End initialization *)
InitOK:=TRUE;
END_ACTION

(* POU Plant_Objects/obj_ZTHL, ST *)
FUNCTION_BLOCK obj_ZTHL
(* === ZIGBEE AMBIENT SENSORS MT-200 ===
   v1.0[07/05/05] - Create
*)
VAR CONSTANT
	(* States *)
	WAIT_STATE			:	BYTE := 0;
	STATUS_REQUEST		:	BYTE := 1;
	LQI_REQUEST			:	BYTE := 2;
	MEAS_REQUEST		:	BYTE := 3;
	END_READ			:	BYTE := 4;
	ERROR_STATE			:	BYTE := 100;

	LQI_Threshold		:	WORD := 100;		(* Zigbee link quality minimum value *)
	LowBattVoltage		:	WORD := 270;		(* Battery is considered low when reaches 1.35V each *)
END_VAR
VAR_INPUT
	(* Settings *)
	ID				: BYTE;
	Address			: BYTE;

	Refresh_Period	: TIME:=t#5m;
	(* Controls *)
	Refresh_Auto	: BOOL:=TRUE; (* Enable automatic refresh *)
	Refresh_Now		: BOOL; 	  (* Force an immediate refresh *)

	(* Limits *)
	Tmin			: INT := 50;
	Tmax			: INT := 400;
END_VAR
VAR_IN_OUT
	(* Interface *)
	MODBUS			: obj_MODBUS_TCP;
END_VAR
VAR_OUTPUT
	OUT_STATUS		: WORD;
	OUT_TEMP		: INT;	(* Temperatura misurata [°C/10] *)
	OUT_HYGRO		: INT;	(* Umidità misurata [%] *)
	OUT_LUX			: INT;	(* Luce misurata [lux] *)
	OUT_VBATT		: INT;	(* Tensione misurata dalla batteria [V/100] *)

	OUT_LQI			: BYTE;

	ERR				: BOOL;

	(* Status *)
	Status_Log		: BYTE;
	Status_Vis 		: DWORD;
END_VAR
VAR
	dly 	 		: TON := (PT:=t#5s);

	sta				: BYTE;
	retry	 		: BYTE;

	Status			: FLT_EVENT;
	Quality			: FLT_EVENT;
	NoSignal		: FLT_EVENT;
	Battery			: FLT_EVENT;
	Temperature		: FLT_EVENT := (INITEV:=FALSE);
	Alarm			: FLT_EVENT;

	AlarmCtr		: BYTE;
	WarningCtr		: BYTE;

	TON_CheckLinkQuality: TON;
	TON_CheckBattery: TON;
END_VAR
CASE sta OF
	WAIT_STATE: (* === Wait update signals *)
		dly(IN:=NOT (dly.Q OR Refresh_Now OR (NOT Refresh_Auto)));
		IF dly.Q OR Refresh_Now THEN
			dly.PT:=Refresh_Period;
			Refresh_Now:=FALSE;
			(*sta:=STATUS_REQUEST;*)
			sta:=LQI_REQUEST;
		END_IF
(*

	STATUS_REQUEST:	(* Node status *)
		IF NOT (MODBUS.MB_Lock OR MODBUS.MB_Start) THEN
			MODBUS.MB_Lock:=TRUE;
			MODBUS.ID:=ID;
			MODBUS.MB_MASTER.bUNIT_ID := Address;
			MODBUS.MB_MASTER.bFUNCTION_CODE:=16#03;
			MODBUS.MB_MASTER.wREAD_ADDRESS:=16#0D;
			MODBUS.MB_MASTER.wREAD_QUANTITY:=16#1;
			MODBUS.MB_Start:=TRUE;
			sta:=LQI_REQUEST;
		END_IF

	LQI_REQUEST:	(* Link quality *)
		IF NOT MODBUS.MB_Start THEN
			IF MODBUS.MB_MASTER.wERROR<>MB_NO_ERROR THEN
				sta:=ERROR_STATE;
			ELSE
				OUT_STATUS	:=	MODBUS.MB_READBUF[0];

				MODBUS.MB_Lock:=TRUE;
				MODBUS.ID:=ID;
				MODBUS.MB_MASTER.bUNIT_ID := Address;
				MODBUS.MB_MASTER.bFUNCTION_CODE:=16#03;
				MODBUS.MB_MASTER.wREAD_ADDRESS:=16#01;
				MODBUS.MB_MASTER.wREAD_QUANTITY:=16#1;
				MODBUS.MB_Start:=TRUE;

				sta:=MEAS_REQUEST;
			END_IF
		END_IF
*)

	LQI_REQUEST:	(* Link quality *)
		IF NOT (MODBUS.MB_Lock OR MODBUS.MB_Start) THEN
				MODBUS.MB_Lock:=TRUE;
				MODBUS.ID:=ID;
				MODBUS.ID:=ID;
				MODBUS.MB_MASTER.bUNIT_ID := Address;
				MODBUS.MB_MASTER.bFUNCTION_CODE:=16#03;
				MODBUS.MB_MASTER.wREAD_ADDRESS:=16#01;
				MODBUS.MB_MASTER.wREAD_QUANTITY:=16#1;
				MODBUS.MB_Start:=TRUE;

				sta:=MEAS_REQUEST;
		END_IF

	MEAS_REQUEST:	(* Measurements *)
		IF NOT MODBUS.MB_Start THEN
			IF MODBUS.MB_MASTER.wERROR<>MB_NO_ERROR THEN
				sta:=ERROR_STATE;
			ELSE

				OUT_LQI	:=	WORD_TO_BYTE(MODBUS.MB_READBUF[0]);

				MODBUS.ID:=ID;
				MODBUS.MB_MASTER.bUNIT_ID := Address;
				MODBUS.MB_MASTER.bFUNCTION_CODE:=16#03;
				MODBUS.MB_MASTER.wREAD_ADDRESS:=16#14;
				MODBUS.MB_MASTER.wREAD_QUANTITY:=16#5;
				MODBUS.MB_Start:=TRUE;

				sta:=END_READ;
			END_IF
		END_IF

	END_READ:	IF NOT MODBUS.MB_Start THEN
			IF MODBUS.MB_MASTER.wERROR<>MB_NO_ERROR THEN
				sta:=ERROR_STATE;
			ELSE
				OUT_TEMP	:=	WORD_TO_INT(MODBUS.MB_READBUF[0]);
				OUT_HYGRO	:=	WORD_TO_INT(MODBUS.MB_READBUF[1]);
				OUT_LUX		:=	WORD_TO_INT(MODBUS.MB_READBUF[2]);
				OUT_VBATT	:=	WORD_TO_INT(MODBUS.MB_READBUF[3]);
				sta:=WAIT_STATE;
				MODBUS.MB_Lock:=FALSE;
			END_IF
		END_IF

	ERROR_STATE:
			MODBUS.MB_Lock:=FALSE;
			(* Retries *)
			retry:=retry+1;
			IF retry>3 THEN
				retry:=0;
				IF Status_Log<>2 THEN
					LogEv(EL_Alarm,EO_ZTHL,ID,4,'');
				END_IF
				Status_Log:=2;
				Status_Vis:=COLOR_RED;
			END_IF
			sta:=WAIT_STATE;

ELSE
			sta:=WAIT_STATE;
END_CASE

(* Check Status *)
Status(IN:=(OUT_STATUS<>1));

IF Status.EVH THEN LogEv(EL_Alarm,EO_ZTHL,ID,3,''); END_IF

(* Check if there is signal (Link Quality different from 0) *)
NoSignal(IN:=(OUT_LQI=0));

IF NoSignal.EVH THEN
	LogEv(EL_Alarm,EO_ZTHL,ID,7,'');
	AlarmCtr := AlarmCtr + 1;
END_IF

IF NoSignal.EVL THEN AlarmCtr := SEL(AlarmCtr=0,AlarmCtr-1,0); END_IF

(* Check Link Quality *)
TON_CheckLinkQuality(IN:=(OUT_LQI < LQI_Threshold) , PT:=t#12h , Q=> , ET=> );
Quality(IN:=(TON_CheckLinkQuality.Q));


IF Quality.EVL THEN
	LogEv(EL_Wrn,EO_ZTHL,ID,2,WORD_TO_STRING(OUT_LQI));
	WarningCtr := WarningCtr + 1;
END_IF

IF Quality.EVH THEN WarningCtr := SEL(WarningCtr=0,WarningCtr-1,0); END_IF

(* If probe (node) is present proceed checking other warnings, otherwise don't transmit anything *)
IF OUT_LQI>0 THEN (* AND OUT_STATUS=1 THEN *)

	(* Check battery voltage *)
TON_CheckBattery(IN:=(OUT_VBATT<LowBattVoltage) , PT:= t#12h, Q=> , ET=> );

	Battery(IN:=TON_CheckBattery.Q);

	IF Battery.EVH THEN
		LogEv(EL_Wrn,EO_ZTHL,ID,6,'');
		WarningCtr := WarningCtr + 1;
	END_IF

	IF Battery.EVL THEN WarningCtr := SEL(WarningCtr=0,WarningCtr-1,0); END_IF

	(* Check Node temperature *)
	Temperature(IN:=(OUT_TEMP<Tmin OR OUT_TEMP>Tmax));

	IF Temperature.EVH THEN
		LogEv(EL_Wrn,EO_ZTHL,ID,5,INT_TO_STRING(OUT_TEMP));
		WarningCtr := WarningCtr + 1;
	END_IF

	IF Temperature.EVL THEN WarningCtr := SEL(WarningCtr=0,WarningCtr-1,0); END_IF

ELSE
	OUT_TEMP 	:= 0;
	OUT_HYGRO 	:= 0;
	OUT_LUX 	:= 0;
	OUT_VBATT 	:= 0;
END_IF

Alarm(IN:=(AlarmCtr=0 AND WarningCtr=0));

IF Alarm.EVH THEN LogEv(EL_Log,EO_ZTHL,ID,1,''); END_IF

IF AlarmCtr>0 THEN
	Status_Log := 2;
	Status_Vis := COLOR_RED;
	ERR := TRUE;
ELSIF WarningCtr>0 THEN
	Status_Log := 1;
	Status_Vis := COLOR_YELLOW;
	ERR := FALSE;
ELSE
	Status_Log := 0;
	Status_Vis := COLOR_GREEN;
	ERR := FALSE;
END_IF
END_FUNCTION_BLOCK
ACTION AddLogData:
Logger.s1:=INSERT('&ZTHL=',BYTE_TO_STRING(ID),5);
IF ID<10 THEN Logger.s1:=INSERT(Logger.s1,'0',5); END_IF

Logger.s1:=CONCAT(Logger.s1,BYTE_TO_STRING(OUT_LQI));			Logger.s1:=CONCAT(Logger.s1,';');
Logger.s1:=CONCAT(Logger.s1,INT_TO_STRING(OUT_TEMP ));			Logger.s1:=CONCAT(Logger.s1,';');
Logger.s1:=CONCAT(Logger.s1,INT_TO_STRING(OUT_HYGRO ));			Logger.s1:=CONCAT(Logger.s1,';');
Logger.s1:=CONCAT(Logger.s1,INT_TO_STRING(OUT_LUX));			Logger.s1:=CONCAT(Logger.s1,';');
Logger.s1:=CONCAT(Logger.s1,INT_TO_STRING(OUT_VBATT));			Logger.s1:=CONCAT(Logger.s1,';');

Logger.s1:=CONCAT(Logger.s1,BYTE_TO_STRING(Status_Log));
ADDSTRING(ADR(Logger.TData), ADR(Logger.s1), Logger.TLen);
END_ACTION

(* POU Utils Functions/PLANT_STATUS, ST *)
FUNCTION_BLOCK PLANT_STATUS
VAR_INPUT
	obj_Status		:	WORD;
END_VAR
VAR_OUTPUT
END_VAR
VAR
	PLANT_STATUS	:	WORD;

	Pwm				:	TON := (PT:=T#1s);
END_VAR
CASE plant_Status OF

	0:	(* Plant OK - Everything works well *)
		(*Pwm(IN:=FALSE);	*)						(* Stop timer if running *)
		LAMP_AL := FALSE;						(* Keep the lamp switched off *)

	(*1:	(* Plant in warning *)
		Pwm(IN:= NOT(Pwm.Q));

		IF Pwm.Q THEN
			LAMP_AL := NOT LAMP_AL;				(* Toggle output *)
		END_IF*)

	2:	(* Plant in alarm *)
		(*Pwm(IN:=FALSE);	*)						(* Stop timer if running *)
		LAMP_AL	:= TRUE;						(* Keep the lamp switched on *)

END_CASE

plant_Status := 0;		(* Reset plant status *)
END_FUNCTION_BLOCK
ACTION UpdateStatus:
IF plant_Status = 2 THEN

	RETURN;					(* If plant already in alarm condition do nothing *)

ELSE

		IF obj_Status <> 0 THEN
			plant_Status := obj_Status;			(* If plant in warning/normal condition and current object in alarm, update plant status *)
		END_IF
END_IF
END_ACTION

(* POU PLC_WDT, ST *)
FUNCTION PLC_WDT: DWORD VAR_INPUT dwEvent: DWORD; dwFilter: DWORD; dwOwner: DWORD; END_VAR
LogEv(EL_AlarmStop,EO_SYS,1,10,'Watchdog');
END_FUNCTION

(* POU Utils Functions/RAW16TOHEXSTR, ST *)
FUNCTION RAW16TOHEXSTR : STRING(128)
VAR_INPUT
	pData: POINTER TO BYTE;
	DataLen: BYTE;
END_VAR
VAR
	pt: POINTER TO BYTE;
	xl: BYTE;
END_VAR
pt:=ADR(RAW16TOHEXSTR);
xl:=0;

WHILE DataLen>0 AND xl<120 DO

	pData:=pData+1;

	pt^ := (pData^ / 16#10) + 48 + (((pData^ / 16#10)/10)*7);
	pt:=pt+1;
	pt^ := (pData^ AND 16#0F)  + 48 + (((pData^ AND 16#0F)/10)*7);
	pt:=pt+1;

	pData:=pData-1;

	pt^ := (pData^ / 16#10) + 48 + (((pData^ / 16#10)/10)*7);
	pt:=pt+1;
	pt^ := (pData^ AND 16#0F)  + 48 + (((pData^ AND 16#0F)/10)*7);
	pt:=pt+1;

	xl:=xl+4;

	DataLen:=DataLen-2;
	pData:=pData+2;

END_WHILE

pt^:=0;
END_FUNCTION

(* POU Utils/RTC_Update, ST *)
FUNCTION RTC_Update : BOOL
VAR
	T: DT;
	TS: STRING;
	TS2: STRING;
	Hour: BYTE;
	Minute: BYTE;
END_VAR
(* Get RTC time *)
T:=SysRtcGetTime(TRUE);
Sys.Time_CT_DT:=T;
(* Calculate variables *)
TS:=DT_TO_STRING(T);
Sys.Time_LogString:=DELETE(STR:=TS, LEN:=3, POS:=1);
TS2:=MID(STR:=TS, LEN:=4, POS:= 4); Sys.Time_Year 	:=STRING_TO_WORD(TS2);
TS2:=MID(STR:=TS, LEN:=2, POS:= 9); Sys.Time_Month	:=STRING_TO_BYTE(TS2);
TS2:=MID(STR:=TS, LEN:=2, POS:=12); Sys.Time_Day  	:=STRING_TO_BYTE(TS2);
Sys.Time_CT_Day:=(32*(Sys.Time_Month-1)+Sys.Time_Day-1);
TS2:=MID(STR:=TS, LEN:=2, POS:=15); Hour			:=STRING_TO_BYTE(TS2);
TS2:=MID(STR:=TS, LEN:=2, POS:=18); Minute		 	:=STRING_TO_BYTE(TS2);
Sys.Time_Hour := Hour;
Sys.Time_Minute := Minute;
Sys.Time_CT_Quarter:=Hour*4+(Minute/15);
END_FUNCTION

(* POU Utils Functions/SHIFT_ARRAY, ST *)
FUNCTION SHIFT_ARRAY : BOOL
VAR_INPUT
	pData	:	POINTER TO ARRAY [1..2] OF WORD;
	Size	:	BYTE;
END_VAR
VAR
	pNew	:	POINTER TO WORD;
	i		:	BYTE;
END_VAR
(* Shift right *)
FOR i:=1 TO (Size-1) BY 1 DO

	(*pNew := pData + 1;*)
	pData^[i] := pData^[i+1];
	(*pData := pData + 1;*)

END_FOR
END_FUNCTION

